(* IEC 61131-3 sources: Yaha/Documentation/Infomaterial/OSCAT/pcworx_basic_333/module_export (part 6) *)

(* ---- SETUP_MONTHS3.ST ---- *)
(*@PROPERTIES_EX@
TYPE: POU
LOCALE: 0
IEC_LANGUAGE: ST
PLC_TYPE: independent
PROC_TYPE: independent
GROUP: SETUP
*)
(*@KEY@:DESCRIPTION*)

(*@KEY@:END_DESCRIPTION*)
FUNCTION_BLOCK SETUP_MONTHS3

(*Group:Default*)

VAR_IN_OUT
	MONTHS3 :	oscat_MONTHS3;
END_VAR

VAR
	init :	BOOL;
END_VAR

(*@KEY@: WORKSHEET
NAME: SETUP_MONTHS3
IEC_LANGUAGE: ST
*)
(* Daten initialisieren *)
IF init THEN RETURN; END_IF;
init := TRUE;

(* ---- english --- *)
MONTHS3[1][01] := 'Jan';
MONTHS3[1][02] := 'Feb';
MONTHS3[1][03] := 'Mar';
MONTHS3[1][04] := 'Apr';
MONTHS3[1][05] := 'May';
MONTHS3[1][06] := 'Jun';
MONTHS3[1][07] := 'Jul';
MONTHS3[1][08] := 'Aug';
MONTHS3[1][09] := 'Sep';
MONTHS3[1][10] := 'Oct';
MONTHS3[1][11] := 'Nov';
MONTHS3[1][12] := 'Dec';

(* ---- german --- *)
MONTHS3[2][01] := 'Jan';
MONTHS3[2][02] := 'Feb';
MONTHS3[2][03] := 'Mrz';
MONTHS3[2][04] := 'Apr';
MONTHs3[2][05] := 'Mai';
MONTHS3[2][06] := 'Jun';
MONTHS3[2][07] := 'Jul';
MONTHS3[2][08] := 'Aug';
MONTHS3[2][09] := 'Sep';
MONTHS3[2][10] := 'Okt';
MONTHS3[2][11] := 'Nov';
MONTHS3[2][12] := 'Dez';

(* ---- french --- *)
MONTHS3[3][01] := 'Jan';
MONTHS3[3][02] := 'Fev';
MONTHS3[3][03] := 'Mar';
MONTHS3[3][04] := 'Avr';
MONTHs3[3][05] := 'Mai';
MONTHS3[3][06] := 'Jun';
MONTHS3[3][07] := 'Jul';
MONTHS3[3][08] := 'Aou';
MONTHS3[3][09] := 'Sep';
MONTHS3[3][10] := 'Oct';
MONTHS3[3][11] := 'Nov';
MONTHS3[3][12] := 'Dec';
(*@KEY@: END_WORKSHEET *)
END_FUNCTION_BLOCK

(* ---- SETUP_WEEKDAYS.ST ---- *)
(*@PROPERTIES_EX@
TYPE: POU
LOCALE: 0
IEC_LANGUAGE: ST
PLC_TYPE: independent
PROC_TYPE: independent
GROUP: SETUP
*)
(*@KEY@:DESCRIPTION*)

(*@KEY@:END_DESCRIPTION*)
FUNCTION_BLOCK SETUP_WEEKDAYS

(*Group:Default*)

VAR_IN_OUT
	WEEKDAYS :	oscat_WEEKDAYS;
END_VAR

VAR
	init :	BOOL;
END_VAR

(*@KEY@: WORKSHEET
NAME: SETUP_WEEKDAYS
IEC_LANGUAGE: ST
*)
(* Daten initialisieren *)
IF init THEN RETURN; END_IF;
init := TRUE;

(* ---- english --- *)
WEEKDAYS[1][01] := 'Monday';
WEEKDAYS[1][02] := 'Tuesday';
WEEKDAYS[1][03] := 'Wednesday';
WEEKDAYS[1][04] := 'Thursday';
WEEKDAYS[1][05] := 'Friday';
WEEKDAYS[1][06] := 'Saturday';
WEEKDAYS[1][07] := 'Sunday';

(* ---- german --- *)
WEEKDAYS[2][01] := 'Montag';
WEEKDAYS[2][02] := 'Dienstag';
WEEKDAYS[2][03] := 'Mittwoch';
WEEKDAYS[2][04] := 'Donnerstag';
WEEKDAYS[2][05] := 'Freitag';
WEEKDAYS[2][06] := 'Samstag';
WEEKDAYS[2][07] := 'Sonntag';

(* ---- french --- *)
WEEKDAYS[3][01] := 'Lundi';
WEEKDAYS[3][02] := 'Mardi';
WEEKDAYS[3][03] := 'Mercredi';
WEEKDAYS[3][04] := 'Jeudi';
WEEKDAYS[3][05] := 'Vendredi';
WEEKDAYS[3][06] := 'Samedi';
WEEKDAYS[3][07] := 'Dimanche';
(*@KEY@: END_WORKSHEET *)
END_FUNCTION_BLOCK

(* ---- SETUP_WEEKDAYS2.ST ---- *)
(*@PROPERTIES_EX@
TYPE: POU
LOCALE: 0
IEC_LANGUAGE: ST
PLC_TYPE: independent
PROC_TYPE: independent
GROUP: SETUP
*)
(*@KEY@:DESCRIPTION*)

(*@KEY@:END_DESCRIPTION*)
FUNCTION_BLOCK SETUP_WEEKDAYS2

(*Group:Default*)

VAR_IN_OUT
	WEEKDAYS2 :	oscat_WEEKDAYS2;
END_VAR

VAR
	init :	BOOL;
END_VAR

(*@KEY@: WORKSHEET
NAME: SETUP_WEEKDAYS2
IEC_LANGUAGE: ST
*)
(* Daten initialisieren *)
IF init THEN RETURN; END_IF;
init := TRUE;

(* ---- english --- *)
WEEKDAYS2[1][01] := 'Mo';
WEEKDAYS2[1][02] := 'Tu';
WEEKDAYS2[1][03] := 'We';
WEEKDAYS2[1][04] := 'Th';
WEEKDAYS2[1][05] := 'Fr';
WEEKDAYS2[1][06] := 'Sa';
WEEKDAYS2[1][07] := 'Su';

(* ---- german --- *)
WEEKDAYS2[2][01] := 'Mo';
WEEKDAYS2[2][02] := 'Di';
WEEKDAYS2[2][03] := 'Mi';
WEEKDAYS2[2][04] := 'Do';
WEEKDAYS2[2][05] := 'Fr';
WEEKDAYS2[2][06] := 'Sa';
WEEKDAYS2[2][07] := 'So';

(* ---- french --- *)
WEEKDAYS2[3][01] := 'Lu';
WEEKDAYS2[3][02] := 'Ma';
WEEKDAYS2[3][03] := 'Me';
WEEKDAYS2[3][04] := 'Je';
WEEKDAYS2[3][05] := 'Ve';
WEEKDAYS2[3][06] := 'Sa';
WEEKDAYS2[3][07] := 'Di';
(*@KEY@: END_WORKSHEET *)
END_FUNCTION_BLOCK

(* ---- SH.ST ---- *)
(*@PROPERTIES_EX@
TYPE: POU
LOCALE: 0
IEC_LANGUAGE: ST
PLC_TYPE: independent
PROC_TYPE: independent
GROUP: ENGINEERING.SIGNAL_PROCESSING
*)
(*@KEY@:DESCRIPTION*)
version 1.1	16 jan 2007
programmer 	hugo
tested by	tobias

this sample and hold module samples an input at the rising edge of clk an stores it in out.
the out stays stable until the next rising clk edge appears.
a trigger output as active for one cycle when the output was updated.
(*@KEY@:END_DESCRIPTION*)
FUNCTION_BLOCK SH

(*Group:Default*)

VAR_INPUT
	IN :	REAL;
	CLK :	BOOL;
END_VAR

VAR_OUTPUT
	OUT :	REAL;
	TRIG :	BOOL;
END_VAR

VAR
	edge :	BOOL;
END_VAR

(*@KEY@: WORKSHEET
NAME: SH
IEC_LANGUAGE: ST
*)
IF clk AND NOT edge THEN
	out := in;
	trig := TRUE;
ELSE;
	trig := FALSE;
END_IF;
edge := clk;

(* revision history

hm 16.1.2007	rev 1.1
	added trig output

*)
(*@KEY@: END_WORKSHEET *)
END_FUNCTION_BLOCK

(* ---- SH_1.ST ---- *)
(*@PROPERTIES_EX@
TYPE: POU
LOCALE: 0
IEC_LANGUAGE: ST
PLC_TYPE: independent
PROC_TYPE: independent
GROUP: ENGINEERING.SIGNAL_PROCESSING
*)
(*@KEY@:DESCRIPTION*)
version 1.2	17 sep 2007
programmer 	hugo
tested by	tobias

this sample and hold module samples an input every PT seconds.
after a ample is taken the output Trig will be active for one cycle.
(*@KEY@:END_DESCRIPTION*)
FUNCTION_BLOCK SH_1

(*Group:Default*)

VAR_INPUT
	IN :	REAL;
	PT :	TIME;
END_VAR

VAR_OUTPUT
	OUT :	REAL;
	TRIG :	BOOL;
END_VAR

VAR
	last :	TIME;
	tx :	TIME;
	T_PLC_MS :	T_PLC_MS;
END_VAR

(*@KEY@: WORKSHEET
NAME: SH_1
IEC_LANGUAGE: ST
*)
(* read system time *)
T_PLC_MS();
tx:= UDINT_TO_TIME(T_PLC_MS.T_PLC_MS);

IF tx - last >= PT THEN
	last := tx;
	out := in;
	trig := TRUE;
ELSE
	trig := FALSE;
END_IF;

(* revision history

HM	6.1.2007	rev 1.1
	added trig output

HM	17.9.2007	rev 1.2
	replaced time() with T_PLC_MS() for compatibility reasons
*)
(*@KEY@: END_WORKSHEET *)
END_FUNCTION_BLOCK

(* ---- SH_2.ST ---- *)
(*@PROPERTIES_EX@
TYPE: POU
LOCALE: 0
IEC_LANGUAGE: ST
PLC_TYPE: independent
PROC_TYPE: independent
GROUP: ENGINEERING.SIGNAL_PROCESSING
*)
(*@KEY@:DESCRIPTION*)
version 1.6	10. mar. 2009
programmer 	hugo
tested by	tobias

this sample and hold module samples an input every PT seconds.
this sample and hold also does avg and other calculations with the input data.
an average is calculated over N samples while for this calculation disc samples are discarded,
disc = 0 all samples are averaged,
if disc = 1 the lowest value is ignored,
if disc = 2 the lowest and highest values are ignored,
and so on.....

(*@KEY@:END_DESCRIPTION*)
FUNCTION_BLOCK SH_2

(*Group:Default*)

VAR_INPUT
	IN :	REAL;
	PT :	TIME;
	N :	INT := INT#16;
	DISC :	INT;
END_VAR

VAR_OUTPUT
	OUT :	REAL;
	TRIG :	BOOL;
	AVG :	REAL;
	HIGH :	REAL;
	LOW :	REAL;
END_VAR

VAR
	M :	INT;
	buf :	oscat_arr_0_15;
	buf2 :	oscat_arr_0_15;
	last :	TIME;
	i :	INT;
	I2 :	INT;
	start :	INT;
	temp :	REAL;
	stop :	INT;
	tx :	TIME;
	d2 :	INT;
	T_PLC_MS :	T_PLC_MS;
END_VAR

(*@KEY@: WORKSHEET
NAME: SH_2
IEC_LANGUAGE: ST
*)
(* read system time *)
T_PLC_MS();
tx:= UDINT_TO_TIME(T_PLC_MS.T_PLC_MS);
d2 := WORD_TO_INT(SHR(INT_TO_WORD(disc),1));

IF tx - last >= PT THEN
	last := tx;
	trig := TRUE;

	(* limit M to 0..16 *)
	M := LIMIT(1,N,16);

	(* edge detected lets take the sample *)
    i := M-1;
    WHILE (i>=1) DO
      i2 := i-1;
      buf2[i] := buf2[i2];
      i:=i-1;
    END_WHILE;

	buf2[0] := in;
	out := in;
	buf := buf2;

	(* sort the ARRAY lowest value AT 0 *)
	FOR start := 0 TO M - 2 DO
		FOR i := start+1 TO M - 1 DO
			IF buf[start] > buf[i] THEN
				temp := buf[start];
				buf[start] := buf[i];
				buf[i] := temp;
			END_IF;
		END_FOR;
	END_FOR;

	(* any calculation with the samples is here *)
	stop := M - 1 - d2;
	start := d2;
	IF NOT even(INT_TO_DINT(disc)) THEN start := start + 1; END_IF;
	avg := 0.0;
	FOR i := start TO stop DO avg := avg + buf[i]; END_FOR;
	avg := avg / INT_TO_REAL(stop - start +1);
	low := buf[start];
	high := buf[stop];
ELSE
	Trig := FALSE;
END_IF;

(* revision history
hm 20. jan. 2007	rev 1.1
	added input N to specify the amout of samples for average and high low calculations
	added trig output

hm 10. sep. 2007 	rev 1.2
	an error would be generated if N was set to 0, now n is forced to1 if set to 0.
	index was out of array.

hm	17. sep. 2007	rev 1.3
	replaced time() with t_plc_ms() for compatibility reasons

hm	6. jan. 2008	rev 1.4
	improved performance

hm	14. jun. 2008	rev 1.5
	set default for input N = 16

hm	10. mar. 2009	rev 1.6
	added type conversion for compatibility reasons

*)
(*@KEY@: END_WORKSHEET *)
END_FUNCTION_BLOCK

(* ---- SH_T.ST ---- *)
(*@PROPERTIES_EX@
TYPE: POU
LOCALE: 0
IEC_LANGUAGE: ST
PLC_TYPE: independent
PROC_TYPE: independent
GROUP: ENGINEERING.SIGNAL_PROCESSING
*)
(*@KEY@:DESCRIPTION*)
version 1.1	18. oct. 2008
programmer 	hugo
tested by	oscat

this sample and hold module samples an input while en is high.
during the high time of en the output follows in.
the out stays stable until the en goes high again.
(*@KEY@:END_DESCRIPTION*)
FUNCTION_BLOCK SH_T

(*Group:Default*)

VAR_INPUT
	IN :	REAL;
	E :	BOOL;
END_VAR

VAR_OUTPUT
	OUT :	REAL;
END_VAR

(*@KEY@: WORKSHEET
NAME: SH_T
IEC_LANGUAGE: ST
*)
IF E THEN out := in; END_IF;

(* revision history
hm	1. sep. 2006	rev 1.0
	original version

hm	18. oct. 2008	rev 1.1
	changed input en to e for compatibility reasons

*)
(*@KEY@: END_WORKSHEET *)
END_FUNCTION_BLOCK

(* ---- SHR_4E.ST ---- *)
(*@PROPERTIES_EX@
TYPE: POU
LOCALE: 0
IEC_LANGUAGE: ST
PLC_TYPE: independent
PROC_TYPE: independent
GROUP: LOGIC.FF_EDGE_TRIGGERED
*)
(*@KEY@:DESCRIPTION*)
version 1.1	25. oct. 2008
programmer 	hugo
tested by	tobias

4 bit shift register with reset
(*@KEY@:END_DESCRIPTION*)
FUNCTION_BLOCK SHR_4E

(*Group:Default*)

VAR_INPUT
	SET :	BOOL;
	D0 :	BOOL;
	CLK :	BOOL;
	RST :	BOOL;
END_VAR

VAR_OUTPUT
	Q0 :	BOOL;
	Q1 :	BOOL;
	Q2 :	BOOL;
	Q3 :	BOOL;
END_VAR

VAR
	trig :	R_TRIG;
END_VAR

(*@KEY@: WORKSHEET
NAME: SHR_4E
IEC_LANGUAGE: ST
*)
(* trig.Q signals a rising edge on clk *)
trig(clk := clk);

IF set OR rst THEN
	Q0 := NOT RST;
	Q1 := Q0;
	Q2 := Q0;
	Q3 := Q0;
ELSIF trig.Q THEN
	Q3 := Q2;
	Q2 := Q1;
	Q1 := Q0;
	Q0 := D0;
END_IF;

(* revision history
hm	4. aug. 2006	rev 1.0
	original version

hm	25. oct. 2008	rev 1.1
	optimized code

*)
(*@KEY@: END_WORKSHEET *)
END_FUNCTION_BLOCK

(* ---- SHR_4UDE.ST ---- *)
(*@PROPERTIES_EX@
TYPE: POU
LOCALE: 0
IEC_LANGUAGE: ST
PLC_TYPE: independent
PROC_TYPE: independent
GROUP: LOGIC.FF_EDGE_TRIGGERED
*)
(*@KEY@:DESCRIPTION*)
version 1.2	14. mar. 2009
programmer 	hugo
tested by	tobias

4 bit shift register with reset up / down direction input
(*@KEY@:END_DESCRIPTION*)
FUNCTION_BLOCK SHR_4UDE

(*Group:Default*)

VAR_INPUT
	SET :	BOOL;
	D0 :	BOOL;
	D3 :	BOOL;
	CLK :	BOOL;
	DN :	BOOL;
	RST :	BOOL;
END_VAR

VAR_OUTPUT
	Q0 :	BOOL;
	Q1 :	BOOL;
	Q2 :	BOOL;
	Q3 :	BOOL;
END_VAR

VAR
	trig :	R_TRIG;
END_VAR

(*@KEY@: WORKSHEET
NAME: SHR_4UDE
IEC_LANGUAGE: ST
*)
(* trig.Q signals a rising edge on clk *)
trig(clk := clk);

IF set OR rst THEN
	Q0 := NOT RST;
	Q1 := Q0;
	Q2 := Q0;
	Q3 := Q0;
ELSIF trig.Q THEN
	IF dn THEN
		Q0 := Q1;
		Q1 := Q2;
		Q2 := Q3;
		Q3 := D3;
	ELSE
		Q3 := Q2;
		Q2 := Q1;
		Q1 := Q0;
		Q0 := D0;
	END_IF;
END_IF;

(* revision history
hm	4. aug. 2006	rev 1.0
	original version

hm	25. oct. 2008	rev 1.1
	optimized code

hm	14. mar. 2009	rev 1.2
	removed double assignments

*)
(*@KEY@: END_WORKSHEET *)
END_FUNCTION_BLOCK

(* ---- SHR_8PLE.ST ---- *)
(*@PROPERTIES_EX@
TYPE: POU
LOCALE: 0
IEC_LANGUAGE: ST
PLC_TYPE: independent
PROC_TYPE: independent
GROUP: LOGIC.FF_EDGE_TRIGGERED
*)
(*@KEY@:DESCRIPTION*)
version 1.0	4 aug 2006
programmer 	hugo
tested by	tobias

8 bit shift register with reset and parallel load
the register can shift up or down
it also has a serial input.
the Din input is on Bit0 for up shift and on bit 7 for down shift
the Dout output is on Bit7 for up shift and on bit 0 for down shift
paralle clock is performed clock synchron while a shift is performed first and then the register is reloaded
(*@KEY@:END_DESCRIPTION*)
FUNCTION_BLOCK SHR_8PLE

(*Group:Default*)

VAR_INPUT
	DIN :	BOOL;
	DLOAD :	BYTE;
	CLK :	BOOL;
	UP :	BOOL := TRUE;
	LOAD :	BOOL;
	RST :	BOOL;
END_VAR

VAR_OUTPUT
	DOUT :	BOOL;
END_VAR

VAR
	edge :	BOOL := TRUE;
	register :	BYTE;
END_VAR

(*@KEY@: WORKSHEET
NAME: SHR_8PLE
IEC_LANGUAGE: ST
*)
(* flankenerkennung clk wird high und edge war high reset ist nicht aktiv und set ist nicht aktiv *)
IF CLK AND edge AND NOT rst THEN
	edge := FALSE;	(* flanke wurde erkannt und weitere flankenerkennung wird verhindert bis edge wieder true ist *)
	(* hier ist der code für das flankenevent *)
	IF UP THEN						(*shift up *)
		register := SHL(register,1);
        register := BIT_LOAD_B(register,Din,0);  (* register.X0 := Din; *)
        Dout     := BIT_OF_DWORD(BYTE_TO_DWORD(register),7);     (* Dout := register.X7; *)
	ELSE						    (* shift down *);
		register := SHR(register,1);
        register := BIT_LOAD_B(register,Din,7);  (* register.X7 := Din; *)
        Dout     := BIT_OF_DWORD(BYTE_TO_DWORD(register),0);     (* Dout := register.X0; *)
	END_IF;
	IF load THEN							(* the byte on Din will be loaded if load = true *)
		register := Dload;
		IF up THEN
            Dout := BIT_OF_DWORD(BYTE_TO_DWORD(register),7); (* register.X7 *)
        ELSE
            Dout := BIT_OF_DWORD(BYTE_TO_DWORD(register),0); (* register.X0 *)
        END_IF;
	END_IF;
END_IF;
IF NOT clk THEN edge := TRUE; END_IF;	(* sobald clk wieder low wird warten auf nächste flanke *)
IF rst THEN									(* wenn reset aktiv dann ausgang rücksetzen *)
	register := BYTE#0;
	Dout := FALSE;
END_IF;
(*@KEY@: END_WORKSHEET *)
END_FUNCTION_BLOCK

(* ---- SHR_8UDE.ST ---- *)
(*@PROPERTIES_EX@
TYPE: POU
LOCALE: 0
IEC_LANGUAGE: ST
PLC_TYPE: independent
PROC_TYPE: independent
GROUP: LOGIC.FF_EDGE_TRIGGERED
*)
(*@KEY@:DESCRIPTION*)
version 1.2	14. mar. 2009
programmer 	hugo
tested by	tobias

8 bit shift register with reset

(*@KEY@:END_DESCRIPTION*)
FUNCTION_BLOCK SHR_8UDE

(*Group:Default*)

VAR_INPUT
	SET :	BOOL;
	D0 :	BOOL;
	D7 :	BOOL;
	CLK :	BOOL;
	DN :	BOOL;
	RST :	BOOL;
END_VAR

VAR_OUTPUT
	Q0 :	BOOL;
	Q1 :	BOOL;
	Q2 :	BOOL;
	Q3 :	BOOL;
	Q4 :	BOOL;
	Q5 :	BOOL;
	Q6 :	BOOL;
	Q7 :	BOOL;
END_VAR

VAR
	trig :	R_TRIG;
END_VAR

(*@KEY@: WORKSHEET
NAME: SHR_8UDE
IEC_LANGUAGE: ST
*)
(* trig.Q signals a rising edge on clk *)
trig(clk := clk);

IF set OR rst THEN
	Q0 := NOT RST;
	Q1 := Q0;
	Q2 := Q0;
	Q3 := Q0;
	Q4 := Q0;
	Q5 := Q0;
	Q6 := Q0;
	Q7 := Q0;
ELSIF trig.Q THEN
	IF dn THEN
		Q0 := Q1;
		Q1 := Q2;
		Q2 := Q3;
		Q3 := Q4;
		Q4 := Q5;
		Q5 := Q6;
		Q6 := Q7;
		Q7 := D7;
	ELSE
		Q7 := Q6;
		Q6 := Q5;
		Q5 := Q4;
		Q4 := Q3;
		Q3 := Q2;
		Q2 := Q1;
		Q1 := Q0;
		Q0 := D0;
	END_IF;
END_IF;

(* revision history
hm	4. aug. 2006	rev 1.0
	original version

hm	25. oct. 2008	rev 1.1
	optimized code

hm	14. mar. 2009	rev 1.2
	removed double assignments

*)
(*@KEY@: END_WORKSHEET *)
END_FUNCTION_BLOCK

(* ---- SIGNAL.ST ---- *)
(*@PROPERTIES_EX@
TYPE: POU
LOCALE: 0
IEC_LANGUAGE: ST
PLC_TYPE: independent
PROC_TYPE: independent
GROUP: ENGINEERING.AUTOMATION
*)
(*@KEY@:DESCRIPTION*)
version 1.0	13 dec 2007
programmer 	hugo
tested by	tobias

this function generates an output signal according to a bit pattern SIG.
the patter is shifted to the output in time steps of TS.
ts defaults to 128 ms if not specified.
(*@KEY@:END_DESCRIPTION*)
FUNCTION_BLOCK SIGNAL

(*Group:Default*)

VAR_INPUT
	IN :	BOOL;
	SIG :	BYTE;
	TS :	TIME;
END_VAR

VAR_OUTPUT
	Q :	BOOL;
END_VAR

VAR
	tx :	DWORD;
	step :	BYTE;
	T_PLC_MS :	T_PLC_MS;
END_VAR

(*@KEY@: WORKSHEET
NAME: SIGNAL
IEC_LANGUAGE: ST
*)
IF in THEN
	(* an alarm is present read system time first *)
    T_PLC_MS();
    tx:= UDINT_TO_DWORD(T_PLC_MS.T_PLC_MS);

	(* calculate the step counter which is the lowest 3 bits of (time / ts) *)
	IF ts > t#0s THEN
		step := DWORD_TO_BYTE(UDINT_TO_DWORD(DWORD_TO_UDINT(tx) / TIME_TO_UDINT(ts)) AND DWORD#16#0000_0007);
	ELSE
		step := DWORD_TO_BYTE(SHR(tx,7) AND DWORD#16#0000_0007);
	END_IF;
	(* convert the value 0-7 in step into one bit only (bit 0-7) *)
	step := SHL(BYTE#1,_BYTE_TO_INT(step));
	(* generate the output signal *)
	Q := (step AND sig) > BYTE#0;
ELSE
	Q := FALSE;
END_IF;

(* revision history
hm	13.12.2007		rev 1.0
	original version

*)
(*@KEY@: END_WORKSHEET *)
END_FUNCTION_BLOCK

(* ---- SIGNAL_4.ST ---- *)
(*@PROPERTIES_EX@
TYPE: POU
LOCALE: 0
IEC_LANGUAGE: ST
PLC_TYPE: independent
PROC_TYPE: independent
GROUP: ENGINEERING.AUTOMATION
*)
(*@KEY@:DESCRIPTION*)
version 1.0	13 dec 2007
programmer 	hugo
tested by	tobias

this function generates one out of 4 signals specified by bit patterns S1 .. S4.
the selected pattern will be shifted with the step time TS.
In1 has higher priority then In2 which has higher priority then IN3 and in4 has the lowest priority.
ts defaults to 128 ms if not specified.
(*@KEY@:END_DESCRIPTION*)
FUNCTION_BLOCK SIGNAL_4

(*Group:Default*)

VAR_INPUT
	IN1 :	BOOL;
	IN2 :	BOOL;
	IN3 :	BOOL;
	IN4 :	BOOL;
	TS :	TIME;
	S1 :	BYTE := 2#1111_1111;
	S2 :	BYTE := 2#1111_0000;
	S3 :	BYTE := 2#1010_1010;
	S4 :	BYTE := 2#1010_0000;
END_VAR

VAR_OUTPUT
	Q :	BOOL;
END_VAR

VAR
	sig :	signal;
END_VAR

(*@KEY@: WORKSHEET
NAME: SIGNAL_4
IEC_LANGUAGE: ST
*)
(* an alarm is present read system time first *)
(* check if an alarm is present if yes set sig to the alarm pattern otherwise exit the routine *)
IF in1 THEN
	sig(in := TRUE, sig := s1, TS := TS);
ELSIF in2 THEN
	sig(in := TRUE, sig := s2, TS := TS);
ELSIF in3 THEN
	sig(in := TRUE, sig := s3, TS := TS);
ELSIF in4 THEN
	sig(in := TRUE, sig := s4, TS := TS);
ELSE
	sig(in := FALSE);
END_IF;

(* set the output *)
Q := sig.Q;

(* revision history
hm	13.12.2007		rev 1.0
	original version

*)
(*@KEY@: END_WORKSHEET *)
END_FUNCTION_BLOCK

(* ---- SPEED.ST ---- *)
(*@PROPERTIES_EX@
TYPE: POU
LOCALE: 0
IEC_LANGUAGE: ST
PLC_TYPE: independent
PROC_TYPE: independent
GROUP: ENGINEERING.CONVERSION
*)
(*@KEY@:DESCRIPTION*)
version 1.1	11. mar. 2009
programmer 	hugo
tested by	oscat

this function converts different speed units
any unused input can simply be left open.
different inputs connected at the same time will be added up.
(*@KEY@:END_DESCRIPTION*)
FUNCTION_BLOCK SPEED

(*Group:Default*)

VAR_INPUT
	MS :	REAL;
	KMH :	REAL;
	KN :	REAL;
	MH :	REAL;
END_VAR

VAR_OUTPUT
	YMS :	REAL;
	YKMH :	REAL;
	YKN :	REAL;
	YMH :	REAL;
END_VAR

(*@KEY@: WORKSHEET
NAME: SPEED
IEC_LANGUAGE: ST
*)
Yms := ms +
		kmh * 0.27777777777778 +
		kn * 0.5144444 +
		mh * 0.44704;
Ykmh := Yms * 3.6;
Ykn := Yms * 1.94384466037535;
Ymh := Yms * 2.23693629205440;

(*
Geschwindigkeit Meter durch Sekunde m/s 1 m/s = 3,6 km/h
km durch (pro) Stunde, nicht „Stundenkilometer“ verwenden
Knoten kn 1 kn = 1 sm/h = 0,5144 m/s

*)
(*@KEY@: END_WORKSHEET *)
END_FUNCTION_BLOCK

(* ---- SRAMP.ST ---- *)
(*@PROPERTIES_EX@
TYPE: POU
LOCALE: 0
IEC_LANGUAGE: ST
PLC_TYPE: independent
PROC_TYPE: independent
GROUP: ENGINEERING.AUTOMATION
*)
(*@KEY@:DESCRIPTION*)
version 1.1	11. mar. 2009
programmer 	hugo
tested by	tobias

RAMPS generates output signal which are slew rate and acceleration controlled.

(*@KEY@:END_DESCRIPTION*)
FUNCTION_BLOCK SRAMP

(*Group:Default*)

VAR_INPUT
	X :	REAL;
	A_UP :	REAL;
	A_DN :	REAL;
	VU_MAX :	REAL;
	VD_MAX :	REAL;
	LIMIT_HIGH :	REAL;
	LIMIT_LOW :	REAL;
	RST :	BOOL;
END_VAR

VAR_OUTPUT
	Y :	REAL;
	V :	REAL;
END_VAR

VAR
	cycle_time :	TC_S;
	init :	BOOL;
END_VAR

(*@KEY@: WORKSHEET
NAME: SRAMP
IEC_LANGUAGE: ST
*)
(* read the system_time in microseconds *)
cycle_time();

(* assure range of inputs *)
A_up := MAX(0.0,A_UP);
A_dn := MIN(0.0,A_dn);
VU_max := MAX(0.0,VU_max);
VD_max := MIN(0.0,VD_MAX);

(* calculate the output offset *)
IF rst OR NOT init THEN
	init := TRUE;
	Y := 0.0;
	V := 0.0;
ELSIF X = Y THEN
	v := 0.0;
ELSIF X > Y THEN
	(* output is too low >> ramp up and brake at the end *)
	(* accelerate the speed and limit to vu_max *)
	v := MIN(v + A_UP * cycle_time.TC, vu_max);
	(* calculate the max speed to be able to brake and select the lowest *)
	v := MIN(SQRT((Y-X) * 2.0 * A_DN), v);
	(* calculate the output and obey limits *)
	y := LIMIT(limit_low, y + MIN(v * cycle_time.TC, X-Y), limit_high);
ELSIF X < Y THEN
	(* output is too high >> ramp dn and brake at the end *)
	(* accelerate the speed and limit to vd_max *)
	v := MAX(v + A_DN * cycle_time.TC, vd_max);
	(* calculate the max speed to be able to brake and select the lowest *)
	v := MAX(-SQRT((Y-X) * 2.0 * A_UP), v);
	(* calculate the output and obey limits *)
	y := LIMIT(limit_low, y + MAX(v * cycle_time.TC, X-Y), limit_high);
END_IF;

(* revision history
hm	13. mar. 2008	rev 1.0
	original version

hm	11. mar. 2009	rev 1.1
	real constants updated to new systax using dot

*)

(*@KEY@: END_WORKSHEET *)
END_FUNCTION_BLOCK

(* ---- STACK_16.ST ---- *)
(*@PROPERTIES_EX@
TYPE: POU
LOCALE: 0
IEC_LANGUAGE: ST
PLC_TYPE: independent
PROC_TYPE: independent
GROUP: LOGIC.MEMORY
*)
(*@KEY@:DESCRIPTION*)
version 2.0	25. jul 2009
programmer 	hugo
tested by	oscat

16 Dword STACK memory

(*@KEY@:END_DESCRIPTION*)
FUNCTION_BLOCK STACK_16

(*Group:Default*)

VAR_INPUT
	DIN :	DWORD;
	E :	BOOL := TRUE;
	RD :	BOOL;
	WD :	BOOL;
	RST :	BOOL;
END_VAR

VAR_OUTPUT
	DOUT :	DWORD;
	EMPTY :	BOOL := TRUE;
	FULL :	BOOL;
END_VAR

VAR
	pt :	INT;
	stack :	oscat_ardw_0_15;
END_VAR

(*@KEY@: WORKSHEET
NAME: STACK_16
IEC_LANGUAGE: ST
*)
IF RST THEN
	(* asynchronous reset for the fifo *)
	pt := 0;
	EMPTY := TRUE;
	FULL := FALSE;
	Dout := DWORD#0;
ELSIF E THEN
	IF NOT EMPTY AND RD THEN
		(* read one element *)
		pt := pt - 1;
		Dout := stack[pt];
		EMPTY := pt = 0;
		FULL := FALSE;
	END_IF;
	IF NOT FULL AND WD THEN
		(* write one element *)
		stack[pt] := Din;
		pt := pt + 1;
		FULL := pt > 15;
		EMPTY := FALSE;
	END_IF;
END_IF;

(* revision history
hm	4. aug. 2006	rev 1.0
	original version

hm	19. feb 2008	rev 1.1
	performance improvements

hm	17. oct. 2008	rev 1.2
	deleted unnecessary init with 0

hm	27. oct. 2008	rev 1.3
	optimized performance

hm	25. jul 2009	rev 2.0
	changed inputs to allow simultsaneous read and write
*)

(*@KEY@: END_WORKSHEET *)
END_FUNCTION_BLOCK

(* ---- STACK_32.ST ---- *)
(*@PROPERTIES_EX@
TYPE: POU
LOCALE: 0
IEC_LANGUAGE: ST
PLC_TYPE: independent
PROC_TYPE: independent
GROUP: LOGIC.MEMORY
*)
(*@KEY@:DESCRIPTION*)
version 2.0	25. jul 2009
programmer 	hugo
tested by	oscat

32 Dword STACK memory
(*@KEY@:END_DESCRIPTION*)
FUNCTION_BLOCK STACK_32

(*Group:Default*)

VAR_INPUT
	DIN :	DWORD;
	E :	BOOL := TRUE;
	RD :	BOOL;
	WD :	BOOL;
	RST :	BOOL;
END_VAR

VAR_OUTPUT
	DOUT :	DWORD;
	EMPTY :	BOOL := TRUE;
	FULL :	BOOL;
END_VAR

VAR
	pt :	INT;
	stack :	oscat_ardw_0_31;
END_VAR

(*@KEY@: WORKSHEET
NAME: STACK_32
IEC_LANGUAGE: ST
*)
IF RST THEN
	(* asynchronous reset for the fifo *)
	pt := 0;
	EMPTY := TRUE;
	FULL := FALSE;
	Dout := DWORD#0;
ELSIF E THEN
	IF NOT EMPTY AND RD THEN
		(* read one element *)
		pt := pt - 1;
		Dout := stack[pt];
		EMPTY := pt = 0;
		FULL := FALSE;
	END_IF;
	IF NOT FULL AND WD THEN
		(* write one element *)
		stack[pt] := Din;
		pt := pt + 1;
		FULL := pt > 31;
		EMPTY := FALSE;
	END_IF;
END_IF;

(* revision history
hm	4. aug. 2006	rev 1.0
	original version

hm	19. feb 2008	rev 1.1
	performance improvements

hm	17. oct. 2008	rev 1.2
	deleted unnecessary init with 0

ks	27. oct. 2008	rev 1.3
	optimized performance

hm	25. jul 2009	rev 2.0
	changed inputs to allow simultsaneous read and write

*)

(*@KEY@: END_WORKSHEET *)
END_FUNCTION_BLOCK

(* ---- STAIR2.ST ---- *)
(*@PROPERTIES_EX@
TYPE: POU
LOCALE: 0
IEC_LANGUAGE: ST
PLC_TYPE: independent
PROC_TYPE: independent
GROUP: ENGINEERING.SIGNAL_PROCESSING
*)
(*@KEY@:DESCRIPTION*)
version 1.4	10. mar. 2009
programmer 	hugo
tested by	oscat

the function stair2 converts an anlog input signal to a staircase like output.
D is the step width for the output signal. the output will use D as a hysteresis for a stairchange.
if D = 0 then the output follows the input without a chage.
(*@KEY@:END_DESCRIPTION*)
FUNCTION_BLOCK STAIR2

(*Group:Default*)

VAR_INPUT
	X :	REAL;
	D :	REAL;
END_VAR

VAR_OUTPUT
	Y :	REAL;
END_VAR

(*@KEY@: WORKSHEET
NAME: STAIR2
IEC_LANGUAGE: ST
*)
IF D > 0.0 THEN
	IF X >= Y + D OR X <= Y - D THEN Y := INT_TO_REAL(FLOOR(X/D)) * D; END_IF;
ELSE
	Y := X;
END_IF;

(* revision history
hm	28 jan 2007		rev 1.0
	original version

hm	27. dec 2007	rev 1.1
	changed code for better performance

hm	30. jun. 2008	rev 1.2
	added type conversions to avoid warnings under codesys 3.0

ks	26. oct. 2008	rev 1.3
	improved code

hm	10. mar. 2009	rev 1.4
	real constants updated to new systax using dot

*)
(*@KEY@: END_WORKSHEET *)
END_FUNCTION_BLOCK

(* ---- STATUS_TO_ESR.ST ---- *)
(*@PROPERTIES_EX@
TYPE: POU
LOCALE: 0
IEC_LANGUAGE: ST
PLC_TYPE: independent
PROC_TYPE: independent
GROUP: OTHER
*)
(*@KEY@:DESCRIPTION*)
version 1.0	6 oct 2006
programmer 	hugo
tested by	tobias

status_to_esr creates esr data from a status byte.
(*@KEY@:END_DESCRIPTION*)
FUNCTION_BLOCK STATUS_TO_ESR

(*Group:Default*)

VAR_INPUT
	STATUS :	BYTE;
	ADRESS :	oscat_STRING10;
	DT_IN :	UDINT;
	TS :	TIME;
END_VAR

VAR_OUTPUT
	STATUS_TO_ESR :	oscat_esr_data;
END_VAR

(*@KEY@: WORKSHEET
NAME: STATUS_TO_ESR
IEC_LANGUAGE: ST
*)
IF status < BYTE#100 THEN
	status_to_ESR.typ := BYTE#1;
ELSIF status < BYTE#200 THEN
	status_to_ESR.typ := BYTE#2;
ELSE
	status_to_ESR.typ := BYTE#3;
END_IF;
status_to_ESR.adress:= adress;
status_to_ESR.DS := DT_in;
status_to_ESR.TS := TS;
status_to_ESR.data[0] := status;
(*@KEY@: END_WORKSHEET *)
END_FUNCTION_BLOCK

(* ---- STORE_8.ST ---- *)
(*@PROPERTIES_EX@
TYPE: POU
LOCALE: 0
IEC_LANGUAGE: ST
PLC_TYPE: independent
PROC_TYPE: independent
GROUP: LOGIC.FF_PULSE_TRIGGERED
*)
(*@KEY@:DESCRIPTION*)
version 1.2	14. mar. 2009
programmer 	hugo
tested by	oscat

Store_4 stores up to 4 boolean inputs until a reset is clearing the outputs.
the respective output is set with a true at the respective input and stays true until a reset is generated.
a set input is used to set all outputs true at the same time, independent of their inputs.
a clear input is used to reset only the lowest priority of the outputs one at a time.
the lowest priority is q3.
(*@KEY@:END_DESCRIPTION*)
FUNCTION_BLOCK STORE_8

(*Group:Default*)

VAR_INPUT
	SET :	BOOL;
	D0 :	BOOL;
	D1 :	BOOL;
	D2 :	BOOL;
	D3 :	BOOL;
	D4 :	BOOL;
	D5 :	BOOL;
	D6 :	BOOL;
	D7 :	BOOL;
	CLR :	BOOL;
	RST :	BOOL;
END_VAR

VAR_OUTPUT
	Q0 :	BOOL;
	Q1 :	BOOL;
	Q2 :	BOOL;
	Q3 :	BOOL;
	Q4 :	BOOL;
	Q5 :	BOOL;
	Q6 :	BOOL;
	Q7 :	BOOL;
END_VAR

VAR
	edge :	BOOL;
END_VAR

(*@KEY@: WORKSHEET
NAME: STORE_8
IEC_LANGUAGE: ST
*)
IF rst OR set THEN
	q0 := NOT rst;
	q1 := q0;
	q2 := q0;
	q3 := q0;
	q4 := q0;
	q5 := q0;
	q6 := q0;
	q7 := q0;
ELSE
	IF D0 THEN Q0 := TRUE; END_IF;
	IF D1 THEN Q1 := TRUE; END_IF;
	IF D2 THEN Q2 := TRUE; END_IF;
	IF D3 THEN Q3 := TRUE; END_IF;
	IF D4 THEN Q4 := TRUE; END_IF;
	IF D5 THEN Q5 := TRUE; END_IF;
	IF D6 THEN Q6 := TRUE; END_IF;
	IF D7 THEN Q7 := TRUE; END_IF;

	IF clr AND NOT edge THEN
		IF q0 THEN q0 := FALSE;
		ELSIF q1 THEN q1 := FALSE;
		ELSIF q2 THEN q2 := FALSE;
		ELSIF q3 THEN q3 := FALSE;
		ELSIF q4 THEN q4 := FALSE;
		ELSIF q5 THEN q5 := FALSE;
		ELSIF q6 THEN q6 := FALSE;
		ELSE q7 := FALSE;
		END_IF;
	END_IF;
	edge := clr;
END_IF;

(* revision history
hm	25.12.2007	rev 1.0
	original version

hm	30. oct. 2008	rev 1.1
	optimized performance

hm	14. mar. 2009	rev 1.2
	removed double assignments

*)

(*@KEY@: END_WORKSHEET *)
END_FUNCTION_BLOCK

(* ---- STRING_TO_TOD.ST ---- *)
(*@PROPERTIES_EX@
TYPE: POU
LOCALE: 0
IEC_LANGUAGE: ST
PLC_TYPE: independent
PROC_TYPE: independent
GROUP: EMULATION
*)
(*@KEY@:DESCRIPTION*)

(*@KEY@:END_DESCRIPTION*)
FUNCTION_BLOCK STRING_TO_TOD

(*Group:Default*)

VAR_INPUT
	_TOD :	STRING;
END_VAR

VAR_OUTPUT
	STRING_TO_TOD :	UDINT;
END_VAR

VAR
	pos :	INT;
	i :	INT;
	tmp :	STRING;
	tmp2 :	STRING;
END_VAR

(*@KEY@: WORKSHEET
NAME: STRING_TO_TOD
IEC_LANGUAGE: ST
*)
(*
TIME_OF_DAY-Konstanten, zum Speichern von Uhrzeiten:

Eine TIME_OF_DAY-Deklaration beginnt mit "tod#", "TOD#", "TIME_OF_DAY#"
oder "time_of_day#", anschließend können Sie eine Uhrzeit angeben in der Schreibweise:
Stunde:Minute:Sekunde. Sekunden können dabei als reelle Zahlen angegeben werden,
es können also auch Sekundenbruchteile angegeben werden.
Mögliche Werte: 00:00:00 bis 23:59:59.999.

Beispiele:

TIME_OF_DAY#15:36:30.123

tod#00:00:00
*)

STRING_TO_TOD := UDINT#0;
i := LEN(_TOD);
pos :=FIND(_TOD,'#');

IF pos>0 AND i>pos THEN
  tmp := RIGHT(_TOD,LEN(_TOD)-pos);
  pos := FIND(tmp,':');
  IF pos>1 THEN
    tmp2 := LEFT(tmp,pos-1);
    tmp := RIGHT(tmp,LEN(tmp)-pos);
    STRING_TO_TOD := STRING_TO_UDINT(tmp2) * UDINT#3600000;

    pos :=FIND(tmp,':');
    IF pos>1 THEN
      tmp2 := LEFT(tmp,pos-1);
      tmp := RIGHT(tmp,LEN(tmp)-pos);
      STRING_TO_TOD := STRING_TO_TOD + STRING_TO_UDINT(tmp2) * UDINT#60000;

      STRING_TO_TOD := STRING_TO_TOD + STRING_TO_UDINT(tmp) * UDINT#1000;
    END_IF;
  END_IF;
END_IF;
(*@KEY@: END_WORKSHEET *)
END_FUNCTION_BLOCK

(* ---- SUN_POS.ST ---- *)
(*@PROPERTIES_EX@
TYPE: POU
LOCALE: 0
IEC_LANGUAGE: ST
PLC_TYPE: independent
PROC_TYPE: independent
GROUP: TIME_DATE
*)
(*@KEY@:DESCRIPTION*)
version 2.1	7. mar. 2009
programmer 	hugo
tested by		oscat

this FUNCTION block calculates the sun position for a given date and time.
the times are calculated in utc and have to be corrected for the given time zone.
B is the angle from north and HR is the highth in degrees.

(*@KEY@:END_DESCRIPTION*)
FUNCTION_BLOCK SUN_POS

(*Group:Default*)

VAR_INPUT
	LATITUDE :	REAL;(*latitude of geographical position*)
	LONGITUDE :	REAL;(*longitude of geographical position*)
	UTC :	UDINT;(*world time*)
END_VAR

VAR_OUTPUT
	B :	REAL;
	HR :	REAL;
END_VAR

VAR
	g :	REAL;
	a :	REAL;
	d :	REAL;
	h :	REAL;
	t1 :	REAL;
	n :	REAL;
	e :	REAL;
	c :	REAL;
	tau :	REAL;
	sin_d :	REAL;
	rlat :	REAL;
	sin_lat :	REAL;
	cos_lat :	REAL;
	cos_tau :	REAL;
	cos_d :	REAL;
	MATH_PI :	REAL := 3.14159265358979323846264338327950288;
	MATH_PI2 :	REAL := 6.28318530717958647692528676655900576;
END_VAR

(*@KEY@: WORKSHEET
NAME: SUN_POS
IEC_LANGUAGE: ST
*)
(* EXIT the routine IF it was executed within 10 seconds which is equal to 0.04 degrees accuracy
depending on startup conditions this could lead to a lockup for 10 seconds and not delivering a usable position
tx := T_PLC_MS();
IF tx - last < 10000 THEN RETURN; END_IF;
last := tx;
*)

(* n is the julian date and the number of days since 1.1.2000-12:00 midday *)
(* be careful for step7 date startes 1.1.1990 instead of 1.1.1970 *)
(* for step7 this line must change *)
n := UDINT_TO_REAL(UTC - UDINT#946728000) * 0.000011574074074074;
g :=MODR(6.240040768 + 0.01720197 * n, MATH_PI2);
d := MODR(4.89495042 + 0.017202792 * n, MATH_PI2) + 0.033423055 * SIN(g) + 0.000349066 * SIN(2.0*g);
e := 0.409087723 - 0.000000006981317008 * n;
cos_d := COS(d);
sin_d := SIN(d);
a := ATAN(COS(e) * sin_d / cos_d);
IF cos_d < 0.0 THEN a := a + MATH_PI; END_IF;
c := ASIN(SIN(e) * sin_d);

(* also here we must be very careful utc is from 1.1.1970 for step7 the formula must change *)
tau := RAD(MODR(6.697376 + (n - 0.25) * 0.0657098245037645 + TOD_TO_REAL(DT_TO_TOD(utc)) * 0.0000002785383333, 24.0) * 15.0 + longitude) - a;
rlat := RAD(latitude);
sin_lat := SIN(rlat);
cos_lat := COS(rlat);
cos_tau := COS(tau);
t1 := cos_tau * sin_lat - TAN(c) * cos_lat;
B := ATAN(SIN(tau) / t1);
IF t1 < 0.0 THEN B := B + MATH_PI2; ELSE B := B + MATH_PI; END_IF;
B := DEG(MODR(B, MATH_PI2));
h := DEG(ASIN(COS(C) * cos_tau * cos_lat +SIN(c) * sin_lat));
IF h > 180.0 THEN h := h - 360.0; END_IF;
(* consider refraction *)
HR := h + REFRACTION(h);

(* revision history
hm	1. feb 2007	rev 1.0
	original version

hm	6. jan 2008	rev 1.1
	performance improvements

hm	18. jan 2008	rev 1.2
	further performance improvements
	only calculate once every 10 seconds

hm	16. mar. 2008	rev 1.3
	added type conversion to avoid warnings under codesys 3.0

hm	30. jun. 2008	rev 1.4
	added type conversions to avoid warnings under codesys 3.0

hm	18. oct. 2008	rev 1.5
	using math constants

hm	17. dec. 2008	rev 1.6
	angles below horizon are displayed in negative degrees

hm	27. feb. 2009	rev 2.0
	new code with better accuracy

hm	7. mar. 2009	rev 2.1
	refraction is added after angle normalization
	deleted 10 second lockout
	added output for astronomical heigth h
*)
(*@KEY@: END_WORKSHEET *)
END_FUNCTION_BLOCK

(* ---- SUN_TIME.ST ---- *)
(*@PROPERTIES_EX@
TYPE: POU
LOCALE: 0
IEC_LANGUAGE: ST
PLC_TYPE: independent
PROC_TYPE: independent
GROUP: TIME_DATE
*)
(*@KEY@:DESCRIPTION*)
version 1.7	25. jan. 2011
programmer 	hugo
tested by	tobias

this FUNCTION block calculates the sun rise, sun set, sun offset at midday sun declination for a given date
for performance reasons the algorithm has been simplified and is accurate within a few minutes only
the times are calculated in utc and have to be corrected for the given time zone
this correction is not done within sun_time because it would be a problem on days where dst is enabled or disabled

(*@KEY@:END_DESCRIPTION*)
FUNCTION_BLOCK SUN_TIME

(*Group:Default*)

VAR_INPUT
	LATITUDE :	REAL;(*latitude of geographical position*)
	LONGITUDE :	REAL;(*longitude of geographical position*)
	UTC :	UDINT;(*world time*)
	H :	REAL := -0.83333333333;(*heighth above horizon for sunrise*)
END_VAR

VAR_OUTPUT
	MIDDAY :	UDINT;(*astrological midday in hours when sun stand at south direction*)
	SUN_RISE :	UDINT;(*sun rise for current day in local time*)
	SUN_SET :	UDINT;(*sun set for current day in local time*)
	SUN_DECLINATION :	REAL;(*sun declination at midday in degrees*)
END_VAR

VAR
	DK :	REAL;(*sun declination at midday*)
	delta :	UDINT;(*delta from midday for sunrise and sunset*)
	B :	REAL;
END_VAR

(*@KEY@: WORKSHEET
NAME: SUN_TIME
IEC_LANGUAGE: ST
*)
B := latitude * 0.0174532925199433;
MIDDAY := SUN_MIDDAY(longitude, utc);
DK := 0.40954 * SIN(0.0172 * (INT_TO_REAL(DAY_OF_YEAR(utc)) - 79.35));
sun_declination := DEG(DK);
IF sun_declination > 180.0 THEN sun_declination := sun_declination - 360.0; END_IF;
sun_declination := 90.0 - LATITUDE + sun_declination;
delta := TIME_TO_UDINT(HOUR_TO_TIME(ACOS((SIN(RAD(H)) - SIN(B) * SIN(DK)) / (COS(B) * COS(DK))) * 3.819718632));
sun_rise := MIDDAY - delta;
sun_set := MIDDAY + delta;

(* revision history

rev 1.1	hm	20.1.2007
	deleted unused variables sun_riseR and sun_setR

rev 1.2 hm 17.4.2007
	corrected error while sun:midday would not be corrected for longitude.

rev 1.3	hm	6. jan 2008
	performance improvements

rev	1.4 hm	17. jan 2008
	calculation is now only performed once a day

hm	10. mar. 2009	rev 1.5
	improved performance
	calculation will be performed on every call to allow movong installations

hm	26. jul 2009	rev 1.6
	fixed a problem with wrong midday calculation

hm	25. jan. 2011	rev 1.7
	using function sun_midday
	corrected angle of sun_declination
	added input H
*)
(*@KEY@: END_WORKSHEET *)
END_FUNCTION_BLOCK

(* ---- T_PLC_MS.ST ---- *)
(*@PROPERTIES_EX@
TYPE: POU
LOCALE: 0
IEC_LANGUAGE: ST
PLC_TYPE: independent
PROC_TYPE: independent
GROUP: ENGINEERING.MEASUREMENTS
*)
(*@KEY@:DESCRIPTION*)
version 1.1	12 nov 2007
programmer 	hugo
tested by	tobias

T_PLC_MS reads the internal PLC timer and return the time, it has the advantage to be able to set a debug mode
and speed up the counter to test the plc timer overrun which occurs every 50 days respectively 25 days at siemens S7
this routine also allows to correct the behavior of s7 where the internal plc counter will not count all 32 bits.
(*@KEY@:END_DESCRIPTION*)
FUNCTION_BLOCK T_PLC_MS

(*Group:Default*)

VAR_OUTPUT
	T_PLC_MS :	UDINT;
END_VAR

VAR_EXTERNAL
	PLC_TICKS_PER_SEC :	INT;(*Systemticks pro Sekunde*)
	PLC_SYS_TICK_CNT :	DINT;(*Anzahl der Systemticks*)
END_VAR

(*Group:Debug-Parameter*)

VAR
	debug :	BOOL;(*Debug-Mode ON / OFF*)
	N :	INT;(*Debug-Faktor*)
	Offset :	UDINT;(*Debug-Offset*)
	temp :	DWORD := DWORD#1;(*Debug-Offset*)
	mode :	BOOL;(*modus*)
	faktor :	UDINT;(*Systemtakt-Faktor*)
	init :	BOOL;
	v_plc_ticks_per_sec :	UDINT;
	base :	UDINT := UDINT#1000;
END_VAR

(*@KEY@: WORKSHEET
NAME: T_PLC_MS
IEC_LANGUAGE: ST
*)
IF init = FALSE THEN
	v_plc_ticks_per_sec := INT_TO_UDINT(PLC_TICKS_PER_SEC);
	IF v_plc_ticks_per_sec = UDINT#1024 THEN
		faktor := UDINT#1;
		mode := FALSE;
	ELSIF v_plc_ticks_per_sec > UDINT#0 THEN
		IF v_plc_ticks_per_sec <= base THEN
			faktor := base / v_plc_ticks_per_sec;
			mode := FALSE;
		ELSE
			faktor := v_plc_ticks_per_sec / base;
			mode := TRUE;
		END_IF;
	ELSE
		faktor := UDINT#1;
	END_IF;
	init := TRUE;
END_IF;

IF mode THEN
	T_PLC_MS := DINT_TO_UDINT(PLC_SYS_TICK_CNT) / faktor;
ELSE
	T_PLC_MS := DINT_TO_UDINT(PLC_SYS_TICK_CNT) * faktor;
END_IF;

IF debug THEN
	T_PLC_MS := (DWORD_TO_UDINT(SHL(UDINT_TO_DWORD(T_PLC_MS),N) OR SHL(temp,N)) - UDINT#1) + Offset;
END_IF;

(* revision history
hm	14.9.2007	rev 1.0
	original version

hm	12. nov 2007	rev 1.1
	added temporaray variable tx because some compilers could not handle time() as an argument

*)
(*@KEY@: END_WORKSHEET *)
END_FUNCTION_BLOCK

(* ---- T_PLC_US.ST ---- *)
(*@PROPERTIES_EX@
TYPE: POU
LOCALE: 0
IEC_LANGUAGE: ST
PLC_TYPE: independent
PROC_TYPE: independent
GROUP: ENGINEERING.MEASUREMENTS
*)
(*@KEY@:DESCRIPTION*)
version 1.1	12 nov 2007
programmer 	hugo
tested by	tobias

T_PLC_US reads the internal PLC timer and return the time, it has the advantage to be able to set a debug mode
and speed up the counter to test the plc timer overrun which occurs every 50 days respectively 25 days at siemens S7
this routine also allows to correct the behavior of s7 where the internal plc counter will not count all 32 bits.
(*@KEY@:END_DESCRIPTION*)
FUNCTION_BLOCK T_PLC_US

(*Group:Default*)

VAR_OUTPUT
	T_PLC_US :	UDINT;
END_VAR

VAR_EXTERNAL
	PLC_TICKS_PER_SEC :	INT;(*Systemticks pro Sekunde*)
	PLC_SYS_TICK_CNT :	DINT;(*Anzahl der Systemticks*)
END_VAR

(*Group:Debug-Parameter*)

VAR
	debug :	BOOL;(*Debug-Mode ON / OFF*)
	N :	INT;(*Debug-Faktor*)
	Offset :	UDINT;(*Debug-Offset*)
	temp :	DWORD := DWORD#1;(*Debug-Offset*)
	mode :	BOOL;(*modus*)
	faktor :	UDINT;(*Systemtakt-Faktor*)
	init :	BOOL;
	v_plc_ticks_per_sec :	UDINT;
	base :	UDINT := UDINT#1000000;
END_VAR

(*@KEY@: WORKSHEET
NAME: T_PLC_US
IEC_LANGUAGE: ST
*)
IF init = FALSE THEN
	v_plc_ticks_per_sec := INT_TO_UDINT(PLC_TICKS_PER_SEC);
	IF v_plc_ticks_per_sec = UDINT#1024 THEN
		faktor := UDINT#1000;
		mode := FALSE;
	ELSIF v_plc_ticks_per_sec > UDINT#0 THEN
		IF v_plc_ticks_per_sec <= base THEN
			faktor := base / v_plc_ticks_per_sec;
			mode := FALSE;
		ELSE
			faktor := v_plc_ticks_per_sec / base;
			mode := TRUE;
		END_IF;
	ELSE
		faktor := UDINT#1;
	END_IF;
	init := TRUE;
END_IF;

IF mode THEN
	T_PLC_US := DINT_TO_UDINT(PLC_SYS_TICK_CNT) / faktor;
ELSE
	T_PLC_US := DINT_TO_UDINT(PLC_SYS_TICK_CNT) * faktor;
END_IF;

IF debug THEN
	T_PLC_US := (DWORD_TO_UDINT(SHL(UDINT_TO_DWORD(T_PLC_US),N) OR SHL(temp,N)) - UDINT#1) + Offset;
END_IF;

(* revision history
hm	14.9.2007	rev 1.0
	original version

hm	12. nov 2007	rev 1.1
	added temporaray variable tx because some compilers could not handle time() as an argument

*)
(*@KEY@: END_WORKSHEET *)
END_FUNCTION_BLOCK

(* ---- TC_MS.ST ---- *)
(*@PROPERTIES_EX@
TYPE: POU
LOCALE: 0
IEC_LANGUAGE: ST
PLC_TYPE: independent
PROC_TYPE: independent
GROUP: ENGINEERING.MEASUREMENTS
*)
(*@KEY@:DESCRIPTION*)
version 1.0	13 mar 2008
programmer 	hugo
tested by	tobias

TC_MS delivers the time it was last called on the output TC in Milliseconds.
(*@KEY@:END_DESCRIPTION*)
FUNCTION_BLOCK TC_MS

(*Group:Default*)

VAR_OUTPUT
	TC :	DWORD;
END_VAR

VAR
	init :	BOOL;
	tx :	UDINT;
	last :	UDINT;
	T_PLC_MS :	T_PLC_MS;
END_VAR

(*@KEY@: WORKSHEET
NAME: TC_MS
IEC_LANGUAGE: ST
*)
(* read system time and prepare input data *)
T_PLC_MS();
tx:= T_PLC_MS.T_PLC_MS;

IF NOT init THEN
	init := TRUE;
	TC := DWORD#0;
ELSE
	tc := UDINT_TO_DWORD(tx - last);
END_IF;
last := tx;

(* revision history
hm		13. mar. 2008	rev 1.0
	original version

*)
(*@KEY@: END_WORKSHEET *)
END_FUNCTION_BLOCK

(* ---- TC_S.ST ---- *)
(*@PROPERTIES_EX@
TYPE: POU
LOCALE: 0
IEC_LANGUAGE: ST
PLC_TYPE: independent
PROC_TYPE: independent
GROUP: ENGINEERING.MEASUREMENTS
*)
(*@KEY@:DESCRIPTION*)
version 1.2	11. mar. 2009
programmer 	hugo
tested by	tobias

TC_S delivers the time it was last called on the output TC in seconds.

(*@KEY@:END_DESCRIPTION*)
FUNCTION_BLOCK TC_S

(*Group:Default*)

VAR_OUTPUT
	TC :	REAL;
END_VAR

VAR
	init :	BOOL;
	tx :	UDINT;
	last :	UDINT;
	T_PLC_US :	T_PLC_US;
END_VAR

(*@KEY@: WORKSHEET
NAME: TC_S
IEC_LANGUAGE: ST
*)
(* read system time and prepare input data *)
T_PLC_US();
tx:= T_PLC_US.T_PLC_US;

IF NOT init THEN
	init := TRUE;
	TC := 0.0;
ELSE
	tc := UDINT_TO_REAL(tx - last) * 1.0E-6;
END_IF;
last := tx;

(* revision history
hm	13. mar. 2008	rev 1.0
	original version

hm	16. mar 2008	rev 1.1
	added type conversion to avoid warnings under codesys 3.0

hm	11. mar. 2009	rev 1.2
	changed real constants to use dot syntax

*)

(*@KEY@: END_WORKSHEET *)
END_FUNCTION_BLOCK

(* ---- TC_US.ST ---- *)
(*@PROPERTIES_EX@
TYPE: POU
LOCALE: 0
IEC_LANGUAGE: ST
PLC_TYPE: independent
PROC_TYPE: independent
GROUP: ENGINEERING.MEASUREMENTS
*)
(*@KEY@:DESCRIPTION*)
version 1.0	13 mar 2008
programmer 	hugo
tested by	tobias

TC_US delivers the time it was last called on the output TC in Microseconds.
(*@KEY@:END_DESCRIPTION*)
FUNCTION_BLOCK TC_US

(*Group:Default*)

VAR_OUTPUT
	TC :	DWORD;
END_VAR

VAR
	init :	BOOL;
	tx :	UDINT;
	last :	UDINT;
	T_PLC_US :	T_PLC_US;
END_VAR

(*@KEY@: WORKSHEET
NAME: TC_US
IEC_LANGUAGE: ST
*)
(* read system time and prepare input data *)
T_PLC_US();
tx:= T_PLC_US.T_PLC_US;

IF NOT init THEN
	init := TRUE;
	TC := DWORD#0;
ELSE
	tc := UDINT_TO_DWORD(tx - last);
END_IF;
last := tx;

(* revision history
hm		13. mar. 2008	rev 1.0
	original version

*)
(*@KEY@: END_WORKSHEET *)
END_FUNCTION_BLOCK

(* ---- TEMPERATURE.ST ---- *)
(*@PROPERTIES_EX@
TYPE: POU
LOCALE: 0
IEC_LANGUAGE: ST
PLC_TYPE: independent
PROC_TYPE: independent
GROUP: ENGINEERING.CONVERSION
*)
(*@KEY@:DESCRIPTION*)
version 1.0	21 feb 2008
programmer 	hugo
tested by	oscat

this function converts different temperature units
any unused input can simply be left open.
different inputs connected at the same time will be added up.
(*@KEY@:END_DESCRIPTION*)
FUNCTION_BLOCK TEMPERATURE

(*Group:Default*)

VAR_INPUT
	K :	REAL;
	C :	REAL := -273.15;
	F :	REAL := -459.67;
	RE :	REAL := -218.52;
	RA :	REAL := 0.0;
END_VAR

VAR_OUTPUT
	YK :	REAL;
	YC :	REAL;
	YF :	REAL;
	YRE :	REAL;
	YRA :	REAL;
END_VAR

(*@KEY@: WORKSHEET
NAME: TEMPERATURE
IEC_LANGUAGE: ST
*)
YK := K + (C + 273.15) + (F + 459.67) * 0.555555555555 + (Re * 1.25 + 273.15) + (Ra * 0.555555555555);
YC := YK -273.15;
YF := YK * 1.8 - 459.67;
YRe := (YK - 273.15) * 0.8;
YRa := YK * 1.8;

(* revision history
hm	21. feb. 2008	rev 1.0
	original version

*)
(*@KEY@: END_WORKSHEET *)
END_FUNCTION_BLOCK

(* ---- TICKER.ST ---- *)
(*@PROPERTIES_EX@
TYPE: POU
LOCALE: 0
IEC_LANGUAGE: ST
PLC_TYPE: independent
PROC_TYPE: independent
GROUP: STRINGS
*)
(*@KEY@:DESCRIPTION*)
version 1.2	29. mar. 2008
programmer 	hugo
tested by	tobias

Ticker sends a substring of text with length N every TD Milliseconds to generate a ticker.
(*@KEY@:END_DESCRIPTION*)
FUNCTION_BLOCK TICKER

(*Group:Default*)

VAR_INPUT
	N :	INT;
	PT :	TIME;
	TEXT :	STRING;
END_VAR

VAR_OUTPUT
	DISPLAY :	STRING;
END_VAR

VAR
	delay :	TP;
	rollout :	STRING;
	text_len :	INT;
	rollout_step :	INT;
	step :	INT;
END_VAR

(*@KEY@: WORKSHEET
NAME: TICKER
IEC_LANGUAGE: ST
*)
(* generate next ticker when delay is low *)
text_len := LEN(text);

IF N < text_len THEN
	IF NOT delay.Q THEN

		IF step > text_len THEN
            rollout_step := 0;
            rollout := '';
            step := 0;
        END_IF;

        IF step + N > text_len THEN
		    (* increase step for next tick *)
		    step := step + 1;
            rollout_step := rollout_step +1;
		    (* extract dispay from text *)
		    display := MID(text, N - rollout_step, step);
            rollout := CONCAT(rollout,'#');
            display := CONCAT(display,rollout);
        ELSE
		    (* increase step for next tick *)
		    step := step + 1;
		    (* extract dispay from text *)
		    display := MID(text, N, step);
        END_IF;

		(* set delay timer for next tick *)
		delay(in := TRUE, PT := PT);
	ELSE;
		(* execute delay timer *)
		delay(in := FALSE);
	END_IF;
ELSE
	display := text;
END_IF;

(* revision history
hm	4. dec. 2007	rev 1.0
	original version

hm	15. dec. 2007	rev 1.1
	step now starts at 1 instaed of 0

hm	29. mar. 2008	rev 1.2
	changed STRING to STRING(STRING_LENGTH)
*)
(*@KEY@: END_WORKSHEET *)
END_FUNCTION_BLOCK

(* ---- TMAX.ST ---- *)
(*@PROPERTIES_EX@
TYPE: POU
LOCALE: 0
IEC_LANGUAGE: ST
PLC_TYPE: independent
PROC_TYPE: independent
GROUP: LOGIC.GENERATORS
*)
(*@KEY@:DESCRIPTION*)
version 1.0	20. jul. 2008
programmer 	hugo
tested by	oscat

Q of tmax will follow IN except that it forces a maximum ontime for the output Q.
the output Z will be active for one cycle if the output is forced low by the timeout.
(*@KEY@:END_DESCRIPTION*)
FUNCTION_BLOCK TMAX

(*Group:Default*)

VAR_INPUT
	IN :	BOOL;
	PT :	TIME;
END_VAR

VAR_OUTPUT
	Q :	BOOL;
	Z :	BOOL;
END_VAR

VAR
	tx :	TIME;
	start :	TIME;
	last_in :	BOOL;
	T_PLC_MS :	T_PLC_MS;
END_VAR

(*@KEY@: WORKSHEET
NAME: TMAX
IEC_LANGUAGE: ST
*)
(* read system timer *)
T_PLC_MS();
tx:= UDINT_TO_TIME(T_PLC_MS.T_PLC_MS);

Z := FALSE;

IF NOT in THEN
	Q := FALSE;
ELSIF IN AND NOT last_in THEN
	Q := TRUE;
	start := tx;
ELSIF (tx - start >= PT) AND Q THEN
	Q := FALSE;
	Z := TRUE;
END_IF;

last_in := IN;

(* revision history
hm	20. jul. 2008	rev 1.0
	original version

*)
(*@KEY@: END_WORKSHEET *)
END_FUNCTION_BLOCK

(* ---- TMIN.ST ---- *)
(*@PROPERTIES_EX@
TYPE: POU
LOCALE: 0
IEC_LANGUAGE: ST
PLC_TYPE: independent
PROC_TYPE: independent
GROUP: LOGIC.GENERATORS
*)
(*@KEY@:DESCRIPTION*)
version 1.0	21. jul. 2008
programmer 	hugo
tested by	oscat

Q of tMIN will follow IN except that it forces a minimum ontime for the output Q.
(*@KEY@:END_DESCRIPTION*)
FUNCTION_BLOCK TMIN

(*Group:Default*)

VAR_INPUT
	IN :	BOOL;
	PT :	TIME;
END_VAR

VAR_OUTPUT
	Q :	BOOL;
END_VAR

VAR
	pm :	TP;
END_VAR

(*@KEY@: WORKSHEET
NAME: TMIN
IEC_LANGUAGE: ST
*)
pm(in := IN, PT := PT);
Q := IN OR pm.Q;

(* revision history
hm	21. jul. 2008	rev 1.0
	original version

*)
(*@KEY@: END_WORKSHEET *)
END_FUNCTION_BLOCK

(* ---- TO_UML.ST ---- *)
(*@PROPERTIES_EX@
TYPE: POU
LOCALE: 0
IEC_LANGUAGE: ST
PLC_TYPE: independent
PROC_TYPE: independent
GROUP: STRINGS
*)
(*@KEY@:DESCRIPTION*)
version 1.1	17. dec. 2008
programmer 		hugo
tested by		tobias

to_uml converts a character above 127 to a two digit character below 127.
the character Ä is converted to Ae
(*@KEY@:END_DESCRIPTION*)
FUNCTION_BLOCK TO_UML

(*Group:Default*)

VAR_INPUT
	IN :	BYTE;
END_VAR

VAR_OUTPUT
	TO_UML :	STRING;
END_VAR

(*@KEY@: WORKSHEET
NAME: TO_UML
IEC_LANGUAGE: ST
*)
CASE _BYTE_TO_INT(in) OF
	196:	(* Ä *)
		TO_UML := 'Ae';
	214:	(* Ö *)
		TO_UML := 'Oe';
	220:	(* Ü *)
		TO_UML := 'Ue';
	223:	(* ß *)
		TO_UML := 'ss';
	228:	(* ä *)
		TO_UML := 'ae';
	246:	(* ö *)
		TO_UML := 'oe';
	252:	(* ü *)
		TO_UML := 'ue';
ELSE
	TO_UML := BYTE_TO_STRING(IN,'%c');
END_CASE;

(* revision history
hm	29. mar. 2008	rev 1.0
	original version

hm	17. dec. 2008	rev 1.1
	changes name of function chr to chr_to_string

*)
(*@KEY@: END_WORKSHEET *)
END_FUNCTION_BLOCK

(* ---- TOD_TO_STRING.ST ---- *)
(*@PROPERTIES_EX@
TYPE: POU
LOCALE: 0
IEC_LANGUAGE: ST
PLC_TYPE: independent
PROC_TYPE: independent
GROUP: EMULATION
*)
(*@KEY@:DESCRIPTION*)

(*@KEY@:END_DESCRIPTION*)
FUNCTION_BLOCK TOD_TO_STRING

(*Group:Default*)

VAR_INPUT
	ITOD :	UDINT;
END_VAR

VAR_OUTPUT
	TOD_STRING :	STRING;
END_VAR

VAR
	st_tmp1 :	STRING;
	st_tmp2 :	STRING;
	cur_hours :	INT;
END_VAR

(*@KEY@: WORKSHEET
NAME: TOD_TO_STRING
IEC_LANGUAGE: ST
*)
cur_hours := hour(ITOD);
IF cur_hours = 0 THEN
  st_tmp2 := '%01dh';
ELSE
  st_tmp2 := '%dh';
END_IF;

st_tmp1 := CONCAT(INT_TO_STRING(cur_hours,st_tmp2),INT_TO_STRING(minute(ITOD),'%02dm'));
TOD_STRING := CONCAT(st_tmp1,UDINT_TO_STRING(ITOD MOD UDINT#60000 / UDINT#1000,'%02us'));
(*@KEY@: END_WORKSHEET *)
END_FUNCTION_BLOCK

(* ---- TOF_1.ST ---- *)
(*@PROPERTIES_EX@
TYPE: POU
LOCALE: 0
IEC_LANGUAGE: ST
PLC_TYPE: independent
PROC_TYPE: independent
GROUP: LOGIC.GENERATORS
*)
(*@KEY@:DESCRIPTION*)
version 1.0	17. jul. 2008
programmer 	hugo
tested by	oscat

TOF_1 will extend a pulse on input in for PT seconds.
in addition the timer can be cleared asynchronously with rst.
TOF_1 is the same function as TOF from the standard LIB except the asynchronous reset input.
(*@KEY@:END_DESCRIPTION*)
FUNCTION_BLOCK TOF_1

(*Group:Default*)

VAR_INPUT
	IN :	BOOL;
	PT :	TIME;
	RST :	BOOL;
END_VAR

VAR_OUTPUT
	Q :	BOOL;
END_VAR

VAR
	start :	TIME;
	tx :	TIME;
	T_PLC_MS :	T_PLC_MS;
END_VAR

(*@KEY@: WORKSHEET
NAME: TOF_1
IEC_LANGUAGE: ST
*)
(* read system timer *)
T_PLC_MS();
tx:= UDINT_TO_TIME(T_PLC_MS.T_PLC_MS);

IF RST THEN
	Q := FALSE;
ELSIF IN THEN
	Q := TRUE;
	start := tx;
ELSIF tx - start >= PT THEN
	Q := FALSE;
END_IF;

(* revision history
hm	17. jul. 2008	rev 1.0
	original version

*)
(*@KEY@: END_WORKSHEET *)
END_FUNCTION_BLOCK

(* ---- TOGGLE.ST ---- *)
(*@PROPERTIES_EX@
TYPE: POU
LOCALE: 0
IEC_LANGUAGE: ST
PLC_TYPE: independent
PROC_TYPE: independent
GROUP: LOGIC.FF_EDGE_TRIGGERED
*)
(*@KEY@:DESCRIPTION*)
version 1.1	30. oct. 2008
programmer 	hugo
tested by	oscat

toggle flip flop the output changes state with every rising edge of clk.
(*@KEY@:END_DESCRIPTION*)
FUNCTION_BLOCK TOGGLE

(*Group:Default*)

VAR_INPUT
	CLK :	BOOL;
	RST :	BOOL;
END_VAR

VAR_OUTPUT
	Q :	BOOL;
END_VAR

VAR
	edge :	BOOL;
END_VAR

(*@KEY@: WORKSHEET
NAME: TOGGLE
IEC_LANGUAGE: ST
*)
IF rst THEN
	Q := FALSE;
ELSIF clk AND NOT edge THEN
	Q := NOT Q;
END_IF;
edge := clk;

(* revision history

hm	13.9.2007		rev 1.0
	original version

hm	30. oct. 2008	rev 1.1
	deleted unnecessary init

*)
(*@KEY@: END_WORKSHEET *)
END_FUNCTION_BLOCK

(* ---- TONOF.ST ---- *)
(*@PROPERTIES_EX@
TYPE: POU
LOCALE: 0
IEC_LANGUAGE: ST
PLC_TYPE: independent
PROC_TYPE: independent
GROUP: LOGIC.GENERATORS
*)
(*@KEY@:DESCRIPTION*)
version 1.2	21. jul 2009
programmer 	hugo
tested by	tobias

TONOF generated a TON and TOF Delay for the Input N TON (T1) and TOF (T2) can be configured separately

(*@KEY@:END_DESCRIPTION*)
FUNCTION_BLOCK TONOF

(*Group:Default*)

VAR_INPUT
	IN :	BOOL;
	T_ON :	TIME;
	T_OFF :	TIME;
END_VAR

VAR_OUTPUT
	Q :	BOOL;
END_VAR

VAR
	X :	TON;
	old :	BOOL;
	mode :	BOOL;
END_VAR

(*@KEY@: WORKSHEET
NAME: TONOF
IEC_LANGUAGE: ST
*)
IF IN XOR old THEN
  X(IN := FALSE, PT := SEL_TIME(IN,T_OFF,T_ON));
  mode := IN;
  old := IN;
END_IF;
X(IN := TRUE);
IF X.Q THEN Q := mode;END_IF;

(* revision history
hm	10. dec 2007	rev 1.0
	original version

hm	17. sep. 2007	rev 1.1
	improved performance

hm	21. jul. 2009	rev 1.2
	fixed a timing probelm

*)

(*@KEY@: END_WORKSHEET *)
END_FUNCTION_BLOCK

(* ---- TP_1.ST ---- *)
(*@PROPERTIES_EX@
TYPE: POU
LOCALE: 0
IEC_LANGUAGE: ST
PLC_TYPE: independent
PROC_TYPE: independent
GROUP: LOGIC.GENERATORS
*)
(*@KEY@:DESCRIPTION*)
version 1.0	28. jun. 2008
programmer 	hugo
tested by	oscat

TP_1 generates a pulse every time it is calles with in := TRUE.
in addition the timer can be cleared asynchronously with rst.
the timer can be retriggered as often as necessary. it will count PT from the last trigger.
(*@KEY@:END_DESCRIPTION*)
FUNCTION_BLOCK TP_1

(*Group:Default*)

VAR_INPUT
	IN :	BOOL;
	PT :	TIME;
	RST :	BOOL;
END_VAR

VAR_OUTPUT
	Q :	BOOL;
END_VAR

VAR
	tx :	TIME;
	start :	TIME;
	ix :	BOOL;
	T_PLC_MS :	T_PLC_MS;
END_VAR

(*@KEY@: WORKSHEET
NAME: TP_1
IEC_LANGUAGE: ST
*)
(* read system timer *)
(* read system_time *)
T_PLC_MS();
tx := UDINT_TO_TIME(T_PLC_MS.T_PLC_MS);

IF RST THEN
	Q := FALSE;
ELSIF IN AND NOT ix THEN
	Q := TRUE;
	start := tx;
ELSIF tx - start >= PT THEN
	Q := FALSE;
END_IF;

ix:= IN;

(* revision history
hm	28. jun. 2008
	original version

*)
(*@KEY@: END_WORKSHEET *)
END_FUNCTION_BLOCK

(* ---- TP_1D.ST ---- *)
(*@PROPERTIES_EX@
TYPE: POU
LOCALE: 0
IEC_LANGUAGE: ST
PLC_TYPE: independent
PROC_TYPE: independent
GROUP: LOGIC.GENERATORS
*)
(*@KEY@:DESCRIPTION*)
version 1.0	28. jun. 2008
programmer 	hugo
tested by	oscat

TP_2 generates a pulse every time it is calles with in := TRUE.
the module will reset IN by itself so no clearing of in is necessary.
in addition the timer can be cleared asynchronously with rst.
also the rst input is cleared by the module itself.
the timer can be retriggered as often as necessary. it will count PT from the last trigger.
after the time PT1 is elapsed, the timer blocks itself for PT2 and only allow new sequences after PT2 has elapsed.
(*@KEY@:END_DESCRIPTION*)
FUNCTION_BLOCK TP_1D

(*Group:Default*)

VAR_INPUT
	IN :	BOOL;
	PT1 :	TIME;
	PTD :	TIME;
	RST :	BOOL;
END_VAR

VAR_OUTPUT
	Q :	BOOL;
	W :	BOOL;
END_VAR

VAR
	tx :	TIME;
	start :	TIME;
	ix :	BOOL;
	T_PLC_MS :	T_PLC_MS;
END_VAR

(*@KEY@: WORKSHEET
NAME: TP_1D
IEC_LANGUAGE: ST
*)
(* read system_time *)
T_PLC_MS();
tx := UDINT_TO_TIME(T_PLC_MS.T_PLC_MS);

IF RST THEN
	Q := FALSE;
	rst := FALSE;
	W := FALSE;
ELSIF W THEN
	IF tx - start >= PTD THEN
		W := FALSE;
	END_IF;
ELSIF IN AND NOT ix THEN
	Q := TRUE;
	start := tx;
	in := FALSE;
ELSIF tx - start >= PT1 THEN
	Q := FALSE;
	W := TRUE;
	start := tx;
END_IF;

ix := IN;

(* revision history
hm	28. jun. 2008
	original version

*)
(*@KEY@: END_WORKSHEET *)
END_FUNCTION_BLOCK

(* ---- TP_X.ST ---- *)
(*@PROPERTIES_EX@
TYPE: POU
LOCALE: 0
IEC_LANGUAGE: ST
PLC_TYPE: independent
PROC_TYPE: independent
GROUP: LOGIC.GENERATORS
*)
(*@KEY@:DESCRIPTION*)
version 1.3	17. dec. 2008
programmer 	hugo
tested by	oscat

retriggerable edge triggered pulse similar to TP but with a retrigger function
if the pt input is 0 then output is always low.
(*@KEY@:END_DESCRIPTION*)
FUNCTION_BLOCK TP_X

(*Group:Default*)

VAR_INPUT
	IN :	BOOL;
	PT :	TIME;
END_VAR

VAR_OUTPUT
	Q :	BOOL;
	ET :	TIME;
END_VAR

VAR
	edge :	BOOL;
	start :	TIME;
	tx :	TIME;
	T_PLC_MS :	T_PLC_MS;
END_VAR

(*@KEY@: WORKSHEET
NAME: TP_X
IEC_LANGUAGE: ST
*)
(* read system_time *)
T_PLC_MS();
tx := UDINT_TO_TIME(T_PLC_MS.T_PLC_MS);

(* rising edge trigger *)
IF IN AND NOT edge THEN
	start := tx;
	Q := PT > t#0ms;
ELSIF Q THEN
	ET := tx - start;
	IF ET >= PT THEN
		Q := FALSE;
		ET := t#0ms;
	END_IF;
END_IF;
edge := IN;

(* revision history
hm	4. aug 2006		rev 1.0
	original version

hm	17. sep 2007	rev 1.1
	replaced time() with T_PLC_MS() for compatibility reasons

hm	19. oct. 2008	rev 1.2
	renamed to TP_R to TP_X for compatibility reasons

hm	17. dec. 2008	rev 1.3
	code optimized

*)
(*@KEY@: END_WORKSHEET *)
END_FUNCTION_BLOCK

(* ---- TREND.ST ---- *)
(*@PROPERTIES_EX@
TYPE: POU
LOCALE: 0
IEC_LANGUAGE: ST
PLC_TYPE: independent
PROC_TYPE: independent
GROUP: ENGINEERING.SIGNAL_PROCESSING
*)
(*@KEY@:DESCRIPTION*)
version 1.0	21. aug. 2009
programmer 	hugo
tested by	oscat

trend analyses the trend of a input signal.
The Output Q is True if the input X is >= last_X and is false if the input X is <= last_X
in addition to the trend the output TU will be high for one cycle to signal a rising of the input value X
and  TD will signal a decreasing value on the input X.
in case of a change the output D will show the delta of the input to the last input value.

(*@KEY@:END_DESCRIPTION*)
FUNCTION_BLOCK TREND

(*Group:Default*)

VAR_INPUT
	X :	REAL;
END_VAR

VAR_OUTPUT
	Q :	BOOL;
	TU :	BOOL;
	TD :	BOOL;
	D :	REAL;
END_VAR

VAR
	last_x :	REAL;
END_VAR

(*@KEY@: WORKSHEET
NAME: TREND
IEC_LANGUAGE: ST
*)
TU := X > last_X;
TD := X < last_X;
Q := TU OR TD;
D := X - LAST_X;

last_X := X;

(* revision history
hm	21. aug. 2009	rev 1.0
	original version

*)

(*@KEY@: END_WORKSHEET *)
END_FUNCTION_BLOCK

(* ---- TREND_DW.ST ---- *)
(*@PROPERTIES_EX@
TYPE: POU
LOCALE: 0
IEC_LANGUAGE: ST
PLC_TYPE: independent
PROC_TYPE: independent
GROUP: ENGINEERING.SIGNAL_PROCESSING
*)
(*@KEY@:DESCRIPTION*)
version 1.2	14. mar. 2009
programmer 	hugo
tested by	oscat

trend_DW analyses the trend of a input signal.
The Output Q is True if the input X is >= last_X and is false if the input X is <= last_X
in addition to the trend the output TU will be high for one cycle to signal a rising of the input value X
and  TD will signal a decreasing value on the input X.
in case of a change the output D will show the delta of the input to the last input value.

(*@KEY@:END_DESCRIPTION*)
FUNCTION_BLOCK TREND_DW

(*Group:Default*)

VAR_INPUT
	X :	DWORD;
END_VAR

VAR_OUTPUT
	Q :	BOOL;
	TU :	BOOL;
	TD :	BOOL;
	D :	DWORD;
END_VAR

VAR
	LAST_X :	DWORD;
END_VAR

(*@KEY@: WORKSHEET
NAME: TREND_DW
IEC_LANGUAGE: ST
*)
IF X > last_X THEN
	TU := TRUE;
	TD := FALSE;
	D := UDINT_TO_DWORD(DWORD_TO_UDINT(X) - DWORD_TO_UDINT(last_X));
	Q := TRUE;
ELSIF X < last_X THEN
	TD := TRUE;
	TU := FALSE;
	D := UDINT_TO_DWORD(DWORD_TO_UDINT(last_X) - DWORD_TO_UDINT(X));
	Q := FALSE;
ELSE
	TU := FALSE;
	TD := FALSE;
	D := DWORD#0;
END_IF;
last_X := X;

(* revision history
hm	21. nov. 2008	rev 1.0
	original version

hm	20. feb. 2009	rev 1.1
	added outputs TU, TD and D

hm	14. mar. 2009	rev 1.2
	removed double assignments

*)

(*@KEY@: END_WORKSHEET *)
END_FUNCTION_BLOCK

(* ---- TRIM.ST ---- *)
(*@PROPERTIES_EX@
TYPE: POU
LOCALE: 0
IEC_LANGUAGE: ST
PLC_TYPE: independent
PROC_TYPE: independent
GROUP: STRINGS
*)
(*@KEY@:DESCRIPTION*)
version 1.2	29. mar. 2008
programmer 	hugo
tested by	tobias

the function deletes all blanks within a string.
(*@KEY@:END_DESCRIPTION*)
FUNCTION_BLOCK TRIM

(*Group:Default*)

VAR_INPUT
	STR :	STRING;
END_VAR

VAR_OUTPUT
	TRIM :	STRING;
END_VAR

VAR
	pos :	INT;
END_VAR

(*@KEY@: WORKSHEET
NAME: TRIM
IEC_LANGUAGE: ST
*)
trim := str;
REPEAT
	pos := FIND(trim,' ');
	IF pos > 0 THEN trim := REPLACE(trim,'',1,pos); END_IF;
UNTIL pos = 0 END_REPEAT;

(* revision histroy
hm	6.10.2006		rev 1.0
	original release

hm	20. mar. 2008	rev 1.1
	avoid to call replace with pos = 0 because some systems will produce an error

hm	29. mar. 2008	rev 1.2
	changed STRING to STRING(STRING_LENGTH)
*)
(*@KEY@: END_WORKSHEET *)
END_FUNCTION_BLOCK

(* ---- TRIM1.ST ---- *)
(*@PROPERTIES_EX@
TYPE: POU
LOCALE: 0
IEC_LANGUAGE: ST
PLC_TYPE: independent
PROC_TYPE: independent
GROUP: STRINGS
*)
(*@KEY@:DESCRIPTION*)
version 1.2	29. mar. 2008
programmer 	hugo
tested by	tobias

the function replaces all multiple blanks within a string by only one blank.
leading and ending blanks will be deleted
(*@KEY@:END_DESCRIPTION*)
FUNCTION_BLOCK TRIM1

(*Group:Default*)

VAR_INPUT
	STR :	STRING;
END_VAR

VAR_OUTPUT
	TRIM1 :	STRING;
END_VAR

VAR
	pos :	INT;
	st_temp :	STRING;
END_VAR

(*@KEY@: WORKSHEET
NAME: TRIM1
IEC_LANGUAGE: ST
*)
trim1 := str;
REPEAT
	pos := FIND(trim1,'  ');
	IF pos > 0 THEN
	  st_temp := trim1;
	  trim1 := REPLACE(trim1,' ',2,pos);
    END_IF;
UNTIL pos = 0 END_REPEAT;
(* beginning and ending blanks need to be stripped off *)
st_temp := LEFT(trim1,1);
IF EQ_STRING(st_temp,' ') THEN trim1 := DELETE(trim1,1,1); END_IF;
st_temp := RIGHT(trim1,1);
IF EQ_STRING(st_temp,' ') THEN trim1 := DELETE(trim1,1,LEN(trim1)); END_IF;

(* revision histroy
hm	4. feb. 2008    rev 1.0
	original release

hm	20. mar. 2008	rev 1.1
	avoid to call replace with pos = 0 because some systems will produce an error

hm	29. mar. 2008	rev 1.2
	changed STRING to STRING(STRING_LENGTH)
*)
(*@KEY@: END_WORKSHEET *)
END_FUNCTION_BLOCK

(* ---- TRIME.ST ---- *)
(*@PROPERTIES_EX@
TYPE: POU
LOCALE: 0
IEC_LANGUAGE: ST
PLC_TYPE: independent
PROC_TYPE: independent
GROUP: STRINGS
*)
(*@KEY@:DESCRIPTION*)
version 1.0	28. mar. 2008
programmer 	hugo
tested by	tobias

this function deletes all leading and ending blanks of a string.
(*@KEY@:END_DESCRIPTION*)
FUNCTION_BLOCK TRIME

(*Group:Default*)

VAR_INPUT
	STR :	STRING;
END_VAR

VAR_OUTPUT
	TRIME :	STRING;
END_VAR

(*@KEY@: WORKSHEET
NAME: TRIME
IEC_LANGUAGE: ST
*)
TRIME := str;
IF LEN(TRIME) < 1 THEN RETURN; END_IF;

WHILE (GET_CHAR(TRIME,1) = 32) DO
	TRIME := DELETE(TRIME,1,1);
END_WHILE;

(* ending blanks need to be stripped off *)
WHILE (GET_CHAR(TRIME,LEN(TRIME)) = 32) DO
	TRIME := DELETE(TRIME,1,LEN(TRIME));
END_WHILE;

(* revision histroy
hm		4. feb. 2008		rev 1.0
	original release

*)
(*@KEY@: END_WORKSHEET *)
END_FUNCTION_BLOCK

(* ---- TUNE.ST ---- *)
(*@PROPERTIES_EX@
TYPE: POU
LOCALE: 0
IEC_LANGUAGE: ST
PLC_TYPE: independent
PROC_TYPE: independent
GROUP: ENGINEERING.AUTOMATION
*)
(*@KEY@:DESCRIPTION*)
version 1.2	11. mar. 2009
programmer 	hugo
tested by	tobias

tune generates an output signal which is set by input switches.
up to 4 switsches can be used to tune the signal up or down.

(*@KEY@:END_DESCRIPTION*)
FUNCTION_BLOCK TUNE

(*Group:Default*)

VAR_INPUT
	SET :	BOOL;
	SU :	BOOL;
	SD :	BOOL;
	RST :	BOOL;
	SS :	REAL := 0.1;
	LIMIT_L :	REAL;
	LIMIT_H :	REAL := 100.0;
	RST_VAL :	REAL;
	SET_VAL :	REAL := 100.0;
	T1 :	TIME := T#500ms;
	T2 :	TIME := T#2s;
	S1 :	REAL := 2.0;
	S2 :	REAL := 10.0;
END_VAR

VAR_OUTPUT
	Y :	REAL;
END_VAR

VAR
	tx :	UDINT;
	start :	UDINT;
	start2 :	UDINT;
	state :	INT;
	in :	BOOL;
	step :	REAL;
	speed :	REAL;
	Y_start :	REAL;
	Y_start2 :	REAL;
	T_PLC_MS :	T_PLC_MS;
END_VAR

(*@KEY@: WORKSHEET
NAME: TUNE
IEC_LANGUAGE: ST
*)
(* read system_time *)
T_PLC_MS();
tx:= T_PLC_MS.T_PLC_MS;

IF rst THEN
	Y := RST_val;
	state := 0;
ELSIF set THEN
	Y := SET_val;
	state := 0;
ELSIF state > 0 THEN
	(* key has been pushed state machine operating *)
	(* first read the correct input *)
	IF state = 1 THEN
		(* step up *)
		in := su;
	ELSE
		(* step down *)
		in := sd;
	END_IF;
	(* check for single step operation *)
	IF NOT in AND tx - start <= TIME_TO_UDINT(T1) THEN
		Y := Y_start + step;
		state := 0;
	(* check if fast ramp needs to be generated *)
	ELSIF in AND tx - start >= TIME_TO_UDINT(T2) THEN
		Y := Y_start2 + UDINT_TO_REAL(tx - start2) * s2 / speed;
	(* check if slow ramp needs to be generated *)
	ELSIF in AND tx - start >= TIME_TO_UDINT(T1) THEN
		Y := Y_start + UDINT_TO_REAL(tx - start - TIME_TO_UDINT(T1)) * S1 / speed;
		start2 := tx;
		Y_start2 := Y;
	ELSIF NOT in THEN
		state := 0;
	END_IF;
ELSIF su THEN
	(* slow step up *)
	state := 1;
	start := tx;
	step := ss;
	speed := 1000.0;
	Y_start := Y;
ELSIF sd THEN
	(* slow step down *)
	state := 2;
	start := tx;
	step := -ss;
	speed := -1000.0;
	Y_start := Y;
END_IF;

(* make sure output does not exceed limits *)
Y := LIMIT(LIMIT_L, Y, LIMIT_H);

(* revision history
hm	3.11.2007		rev 1.0
	original version

hm	16. mar. 2008	rev 1.1
	added type conversions to avoid warnings under codesys 3.0

hm	11. mar. 2009	rev 1.2
	real constants updated to new systax using dot

*)
(*@KEY@: END_WORKSHEET *)
END_FUNCTION_BLOCK

(* ---- TUNE2.ST ---- *)
(*@PROPERTIES_EX@
TYPE: POU
LOCALE: 0
IEC_LANGUAGE: ST
PLC_TYPE: independent
PROC_TYPE: independent
GROUP: ENGINEERING.AUTOMATION
*)
(*@KEY@:DESCRIPTION*)
version 1.2	11. mar. 2009
programmer 	hugo
tested by	tobias

tune2 generates an output signal which is set by input switches.
up to 4 switsches can be used to tune the signal up or down.

(*@KEY@:END_DESCRIPTION*)
FUNCTION_BLOCK TUNE2

(*Group:Default*)

VAR_INPUT
	SET :	BOOL;
	SU :	BOOL;
	SD :	BOOL;
	FU :	BOOL;
	FD :	BOOL;
	RST :	BOOL;
	SS :	REAL := 0.1;
	FS :	REAL := 5.0;
	LIMIT_L :	REAL;
	LIMIT_H :	REAL := 100.0;
	RST_VAL :	REAL;
	SET_VAL :	REAL := 100.0;
	TR :	TIME := T#500ms;
	S1 :	REAL := 2.0;
	S2 :	REAL := 10.0;
END_VAR

VAR_OUTPUT
	Y :	REAL;
END_VAR

VAR
	tx :	UDINT;
	start :	UDINT;
	state :	INT;
	in :	BOOL;
	step :	REAL;
	speed :	REAL;
	Y_start :	REAL;
	T_PLC_MS :	T_PLC_MS;
END_VAR

(*@KEY@: WORKSHEET
NAME: TUNE2
IEC_LANGUAGE: ST
*)
(* read system time *)
T_PLC_MS();
tx:= T_PLC_MS.T_PLC_MS;

IF rst THEN
	Y := RST_val;
	state := 0;
ELSIF set THEN
	Y := SET_val;
	state := 0;
ELSIF state > 0 THEN
	(* key has been pushed state machine operating *)
	(* first read the correct input *)
	CASE state OF
		1 :	(* slow up *)
			in := su;
		2 :	(* slow down *)
			in := sd;
		3 :	(* fast up *)
			in := fu;
		4 :	(* fast down *)
			in := fd;
	END_CASE;
	(* check for single step operation *)
	IF NOT in AND tx - start <= TIME_TO_UDINT(TR) THEN
		Y := Y_start + step;
		state := 0;
	(* check if ramp needs to be generated *)
	ELSIF in AND tx - start >= TIME_TO_UDINT(TR) THEN
		Y := Y_start + UDINT_TO_REAL(tx - start - TIME_TO_UDINT(TR)) * speed;
	ELSIF NOT in THEN
		state := 0;
	END_IF;
ELSIF su THEN
	(* slow step up *)
	state := 1;
	start := tx;
	step := ss;
	speed := s1 * 1.0E-3;
	Y_start := Y;
ELSIF sd THEN
	(* slow step down *)
	state := 2;
	start := tx;
	step := -ss;
	speed := -s1 * 1.0E-3;
	Y_start := Y;
ELSIF fu THEN
	(* fast step up *)
	state := 3;
	start := tx;
	step := fs;
	speed := s2 * 1.0E-3;
	y_start := Y;
ELSIF fd THEN
	(* fast step down *)
	state := 4;
	start := tx;
	step := -fs;
	speed := -s2 * 1.0E-3;
	y_start := Y;
END_IF;

(* make sure output does not exceed limits *)
Y := LIMIT(LIMIT_L, Y, LIMIT_H);

(* revision history
hm	3.11.2007		rev 1.0
	original version

hm	16. 3. 2008	rev 1.1
	added type conversions to avoid warnings in codesys 3.0
	improved performance

hm	11. mar. 2009	rev 1.2
	real constants updated to new systax using dot

*)
(*@KEY@: END_WORKSHEET *)
END_FUNCTION_BLOCK

(* ---- UPPERCASE.ST ---- *)
(*@PROPERTIES_EX@
TYPE: POU
LOCALE: 0
IEC_LANGUAGE: ST
PLC_TYPE: independent
PROC_TYPE: independent
GROUP: STRINGS
*)
(*@KEY@:DESCRIPTION*)
version 1.3	29. mar. 2008
programmer 	hugo
tested by	tobias

uppercase returns str while all letters a..z and ä,ö,ü are converted to uppercase
(*@KEY@:END_DESCRIPTION*)
FUNCTION_BLOCK UPPERCASE

(*Group:Default*)

VAR_INPUT
	STR :	STRING;
END_VAR

VAR_OUTPUT
	UPPERCASE :	STRING;
END_VAR

VAR
	char :	BYTE;
	char2 :	BYTE;
	pos :	INT;
	l :	INT;
	str_temp :	STRING;
END_VAR

(*@KEY@: WORKSHEET
NAME: UPPERCASE
IEC_LANGUAGE: ST
*)
UPPERCASE := str;
l := LEN(str);
FOR pos := 1 TO l DO
    char := INT_TO_BYTE(GET_CHAR(str,pos));
	char2 := TO_UPPER(char);
    IF char <> char2 THEN
    	str_temp := UPPERCASE;
      	UPPERCASE := REPLACE(str_temp,BYTE_TO_STRING(char2,'%c'),1,pos);
	END_IF;
END_FOR;

(* revision histroy
hm	6. oct. 2006	rev 1.0
	original release

hm	4. feb. 2008	rev 1.1
	improved performance
	added Ä,Ö,Ü

hm	6. mar. 2008	rev 1.2
	added support for exteded Ascii

hm	29. mar. 2008	rev 1.3
	changed STRING to STRING(STRING_LENGTH)
*)
(*@KEY@: END_WORKSHEET *)
END_FUNCTION_BLOCK

(* ---- V3_ABS.ST ---- *)
(*@PROPERTIES_EX@
TYPE: POU
LOCALE: 0
IEC_LANGUAGE: ST
PLC_TYPE: independent
PROC_TYPE: independent
GROUP: MATHEMATICAL.VEKTORMATHEMATIK
*)
(*@KEY@:DESCRIPTION*)
version 1.0	11 dec 2007
programmer 	hugo
tested by	tobias

this function calculates the length of a vectors in a 3 dimensional space
(*@KEY@:END_DESCRIPTION*)
FUNCTION_BLOCK V3_ABS

(*Group:Default*)

VAR_INPUT
	A :	oscat_vector_3;
END_VAR

VAR_OUTPUT
	V3_ABS :	REAL;
END_VAR

(*@KEY@: WORKSHEET
NAME: V3_ABS
IEC_LANGUAGE: ST
*)
V3_ABS := SQRT(A.X * A.X + A.Y * A.Y + A.Z * A.Z);

(* revision history
hm		11 dec 2007	rev 1.0
	original version

*)
(*@KEY@: END_WORKSHEET *)
END_FUNCTION_BLOCK

(* ---- V3_ADD.ST ---- *)
(*@PROPERTIES_EX@
TYPE: POU
LOCALE: 0
IEC_LANGUAGE: ST
PLC_TYPE: independent
PROC_TYPE: independent
GROUP: MATHEMATICAL.VEKTORMATHEMATIK
*)
(*@KEY@:DESCRIPTION*)
version 1.0	11 dec 2007
programmer 	hugo
tested by	tobias

this function adds two vectors in a 3 dimensional space
(*@KEY@:END_DESCRIPTION*)
FUNCTION_BLOCK V3_ADD

(*Group:Default*)

VAR_INPUT
	A :	oscat_vector_3;
	B :	oscat_vector_3;
END_VAR

VAR_OUTPUT
	V3_ADD :	oscat_vector_3;
END_VAR

(*@KEY@: WORKSHEET
NAME: V3_ADD
IEC_LANGUAGE: ST
*)
V3_ADD.X := A.X + B.X;
V3_ADD.Y := A.Y + B.Y;
V3_ADD.Z := A.Z + B.Z;

(* revision history
hm		11 dec 2007	rev 1.0
	original version

*)
(*@KEY@: END_WORKSHEET *)
END_FUNCTION_BLOCK

(* ---- V3_ANG.ST ---- *)
(*@PROPERTIES_EX@
TYPE: POU
LOCALE: 0
IEC_LANGUAGE: ST
PLC_TYPE: independent
PROC_TYPE: independent
GROUP: MATHEMATICAL.VEKTORMATHEMATIK
*)
(*@KEY@:DESCRIPTION*)
version 1.1	10. mar. 2009
programmer 	hugo
tested by	tobias

this function calculates the angle between two vectors in a 3 dimensional space

(*@KEY@:END_DESCRIPTION*)
FUNCTION_BLOCK V3_ANG

(*Group:Default*)

VAR_INPUT
	A :	oscat_vector_3;
	B :	oscat_vector_3;
END_VAR

VAR_OUTPUT
	V3_ANG :	REAL;
END_VAR

VAR
	d :	REAL;
	V3_ABS :	V3_ABS;
	V3_DPRO :	V3_DPRO;
END_VAR

(*@KEY@: WORKSHEET
NAME: V3_ANG
IEC_LANGUAGE: ST
*)

V3_ABS(A:=A);
d :=V3_ABS.V3_ABS;

V3_ABS(A:=B);
d := d * V3_ABS.V3_ABS;

IF d > 0.0 THEN
    V3_DPRO(A:=A,B:=B);
	V3_ANG := ACOS(LIMIT(-1.0, V3_DPRO.V3_DPRO / d,1.0));
ELSE
    V3_ANG := 0.0;

END_IF;

(* revision history
hm	11. dec. 2007	rev 1.0
	original version

hm	10. mar. 2009	rev 1.1
	changed syntax of real constants to 0.0

*)
(*@KEY@: END_WORKSHEET *)
END_FUNCTION_BLOCK

(* ---- V3_DPRO.ST ---- *)
(*@PROPERTIES_EX@
TYPE: POU
LOCALE: 0
IEC_LANGUAGE: ST
PLC_TYPE: independent
PROC_TYPE: independent
GROUP: MATHEMATICAL.VEKTORMATHEMATIK
*)
(*@KEY@:DESCRIPTION*)
version 1.0	11 dec 2007
programmer 	hugo
tested by	tobias

this function calculates the dot product of two vectors in 3 dimensional space
(*@KEY@:END_DESCRIPTION*)
FUNCTION_BLOCK V3_DPRO

(*Group:Default*)

VAR_INPUT
	A :	oscat_vector_3;
	B :	oscat_vector_3;
END_VAR

VAR_OUTPUT
	V3_DPRO :	REAL;
END_VAR

(*@KEY@: WORKSHEET
NAME: V3_DPRO
IEC_LANGUAGE: ST
*)
V3_DPRO := A.X * B.X + A.Y * B.Y + A.Z * B.Z;

(* revision history
hm		11 dec 2007	rev 1.0
	original version

*)
(*@KEY@: END_WORKSHEET *)
END_FUNCTION_BLOCK

(* ---- V3_NORM.ST ---- *)
(*@PROPERTIES_EX@
TYPE: POU
LOCALE: 0
IEC_LANGUAGE: ST
PLC_TYPE: independent
PROC_TYPE: independent
GROUP: MATHEMATICAL.VEKTORMATHEMATIK
*)
(*@KEY@:DESCRIPTION*)
version 1.1	10. mar. 2009
programmer 	hugo
tested by	tobias

this function generates a vectors with absolute length 1 from a vector A in a 3 dimensional space

(*@KEY@:END_DESCRIPTION*)
FUNCTION_BLOCK V3_NORM

(*Group:Default*)

VAR_INPUT
	A :	oscat_vector_3;
END_VAR

VAR_OUTPUT
	V3_NORM :	oscat_vector_3;
END_VAR

VAR
	la :	REAL;
	V3_SMUL :	V3_SMUL;
	V3_ABS :	V3_ABS;
END_VAR

(*@KEY@: WORKSHEET
NAME: V3_NORM
IEC_LANGUAGE: ST
*)

V3_ABS(A:=A);
la:=V3_ABS.V3_ABS;

IF la > 0.0 THEN
    V3_SMUL(A:=A,M:=1.0/la);
    V3_NORM:=V3_SMUL.V3_SMUL;
ELSE
    V3_NORM.X := 0.0;
    V3_NORM.Y := 0.0;
    V3_NORM.Z := 0.0;
END_IF;

(* revision history
hm	11 dec 2007	rev 1.0
	original version

hm	10. mar. 2009	rev 1.1
	changed syntax of real constants to 0.0

*)
(*@KEY@: END_WORKSHEET *)
END_FUNCTION_BLOCK

(* ---- V3_NUL.ST ---- *)
(*@PROPERTIES_EX@
TYPE: POU
LOCALE: 0
IEC_LANGUAGE: ST
PLC_TYPE: independent
PROC_TYPE: independent
GROUP: MATHEMATICAL.VEKTORMATHEMATIK
*)
(*@KEY@:DESCRIPTION*)
version 1.1	10. mar. 2009
programmer 	hugo
tested by	tobias

this function checks if a vectors in a null Vector
(*@KEY@:END_DESCRIPTION*)
FUNCTION_BLOCK V3_NUL

(*Group:Default*)

VAR_INPUT
	A :	oscat_vector_3;
END_VAR

VAR_OUTPUT
	V3_NUL :	BOOL;
END_VAR

(*@KEY@: WORKSHEET
NAME: V3_NUL
IEC_LANGUAGE: ST
*)
V3_NUL := A.X = 0.0 AND A.Y = 0.0 AND A.Z = 0.0;

(* revision history
hm	12 dec 2007	rev 1.0
	original version

hm	10. mar. 2009	rev 1.1
	changed syntax of real constants to 0.0

*)
(*@KEY@: END_WORKSHEET *)
END_FUNCTION_BLOCK

(* ---- V3_PAR.ST ---- *)
(*@PROPERTIES_EX@
TYPE: POU
LOCALE: 0
IEC_LANGUAGE: ST
PLC_TYPE: independent
PROC_TYPE: independent
GROUP: MATHEMATICAL.VEKTORMATHEMATIK
*)
(*@KEY@:DESCRIPTION*)
version 1.1	10. mar. 2009
programmer 	hugo
tested by	tobias

this function checks if two vectors in a 3 dimensional space are parallel.
which means the two vectors have the same direction
(*@KEY@:END_DESCRIPTION*)
FUNCTION_BLOCK V3_PAR

(*Group:Default*)

VAR_INPUT
	A :	oscat_vector_3;
	B :	oscat_vector_3;
END_VAR

VAR_OUTPUT
	V3_PAR :	BOOL;
END_VAR

VAR
	V3_XPRO :	V3_XPRO;
	V3_ABS :	V3_ABS;
END_VAR

(*@KEY@: WORKSHEET
NAME: V3_PAR
IEC_LANGUAGE: ST
*)
V3_XPRO(A:=A,B:=B);
V3_ABS(A:=V3_XPRO.V3_XPRO);

V3_PAR := V3_ABS.V3_ABS = 0.0;

(* revision history
hm	11 dec 2007	rev 1.0
	original version

hm	10. mar. 2009	rev 1.1
	changed syntax of real constants to 0.0

*)
(*@KEY@: END_WORKSHEET *)
END_FUNCTION_BLOCK

(* ---- V3_REV.ST ---- *)
(*@PROPERTIES_EX@
TYPE: POU
LOCALE: 0
IEC_LANGUAGE: ST
PLC_TYPE: independent
PROC_TYPE: independent
GROUP: MATHEMATICAL.VEKTORMATHEMATIK
*)
(*@KEY@:DESCRIPTION*)
version 1.0	11 dec 2007
programmer 	hugo
tested by	tobias

this function reverses a vector in a 3 dimensional space
(*@KEY@:END_DESCRIPTION*)
FUNCTION_BLOCK V3_REV

(*Group:Default*)

VAR_INPUT
	A :	oscat_vector_3;
END_VAR

VAR_OUTPUT
	V3_REV :	oscat_vector_3;
END_VAR

(*@KEY@: WORKSHEET
NAME: V3_REV
IEC_LANGUAGE: ST
*)
V3_REV.X := -A.X;
V3_REV.Y := -A.Y;
V3_REV.Z := -A.Z;

(* revision history
hm		11 dec 2007	rev 1.0
	original version

*)
(*@KEY@: END_WORKSHEET *)
END_FUNCTION_BLOCK

(* ---- V3_SMUL.ST ---- *)
(*@PROPERTIES_EX@
TYPE: POU
LOCALE: 0
IEC_LANGUAGE: ST
PLC_TYPE: independent
PROC_TYPE: independent
GROUP: MATHEMATICAL.VEKTORMATHEMATIK
*)
(*@KEY@:DESCRIPTION*)
version 1.0	11 dec 2007
programmer 	hugo
tested by	tobias

this function multiplies a vectors in a 3 dimensional space with a skalar M
(*@KEY@:END_DESCRIPTION*)
FUNCTION_BLOCK V3_SMUL

(*Group:Default*)

VAR_INPUT
	A :	oscat_vector_3;
	M :	REAL;
END_VAR

VAR_OUTPUT
	V3_SMUL :	oscat_vector_3;
END_VAR

(*@KEY@: WORKSHEET
NAME: V3_SMUL
IEC_LANGUAGE: ST
*)
V3_SMUL.X := A.X * M;
V3_SMUL.Y := A.Y * M;
V3_SMUL.Z := A.Z * M;

(* revision history
hm		11 dec 2007	rev 1.0
	original version

*)
(*@KEY@: END_WORKSHEET *)
END_FUNCTION_BLOCK

(* ---- V3_SUB.ST ---- *)
(*@PROPERTIES_EX@
TYPE: POU
LOCALE: 0
IEC_LANGUAGE: ST
PLC_TYPE: independent
PROC_TYPE: independent
GROUP: MATHEMATICAL.VEKTORMATHEMATIK
*)
(*@KEY@:DESCRIPTION*)
version 1.0	11 dec 2007
programmer 	hugo
tested by	tobias

this function subtracts two vectors in a 3 dimensional space
V3_SUB = A - B
(*@KEY@:END_DESCRIPTION*)
FUNCTION_BLOCK V3_SUB

(*Group:Default*)

VAR_INPUT
	A :	oscat_vector_3;
	B :	oscat_vector_3;
END_VAR

VAR_OUTPUT
	V3_SUB :	oscat_vector_3;
END_VAR

(*@KEY@: WORKSHEET
NAME: V3_SUB
IEC_LANGUAGE: ST
*)
V3_SUB.X := A.X - B.X;
V3_SUB.Y := A.Y - B.Y;
V3_SUB.Z := A.Z - B.Z;

(* revision history
hm		11 dec 2007	rev 1.0
	original version

*)
(*@KEY@: END_WORKSHEET *)
END_FUNCTION_BLOCK

(* ---- V3_XANG.ST ---- *)
(*@PROPERTIES_EX@
TYPE: POU
LOCALE: 0
IEC_LANGUAGE: ST
PLC_TYPE: independent
PROC_TYPE: independent
GROUP: MATHEMATICAL.VEKTORMATHEMATIK
*)
(*@KEY@:DESCRIPTION*)
version 1.1	10. mar. 2009
programmer 	hugo
tested by	tobias

this function calculates the angle between the X-axis and a vectors in a 3 dimensional space

(*@KEY@:END_DESCRIPTION*)
FUNCTION_BLOCK V3_XANG

(*Group:Default*)

VAR_INPUT
	A :	oscat_vector_3;
END_VAR

VAR_OUTPUT
	V3_XANG :	REAL;
END_VAR

VAR
	la :	REAL;
	V3_ABS :	V3_ABS;
END_VAR

(*@KEY@: WORKSHEET
NAME: V3_XANG
IEC_LANGUAGE: ST
*)

V3_ABS(A:=A);
la:=V3_ABS.V3_ABS;

IF la > 0.0 THEN
	V3_XANG := ACOS(A.X / la);
ELSE
    V3_XANG := 0.0;
END_IF;

(* revision history
hm	11 dec 2007	rev 1.0
	original version

hm	10. mar. 2009	rev 1.1
	changed syntax of real constants to 0.0

*)
(*@KEY@: END_WORKSHEET *)
END_FUNCTION_BLOCK

(* ---- V3_XPRO.ST ---- *)
(*@PROPERTIES_EX@
TYPE: POU
LOCALE: 0
IEC_LANGUAGE: ST
PLC_TYPE: independent
PROC_TYPE: independent
GROUP: MATHEMATICAL.VEKTORMATHEMATIK
*)
(*@KEY@:DESCRIPTION*)
version 1.0	11 dec 2007
programmer 	hugo
tested by	tobias

this function adds two vectors in a 3 dimensional space
(*@KEY@:END_DESCRIPTION*)
FUNCTION_BLOCK V3_XPRO

(*Group:Default*)

VAR_INPUT
	A :	oscat_vector_3;
	B :	oscat_vector_3;
END_VAR

VAR_OUTPUT
	V3_XPRO :	oscat_vector_3;
END_VAR

(*@KEY@: WORKSHEET
NAME: V3_XPRO
IEC_LANGUAGE: ST
*)
V3_XPRO.X := A.Y * B.Z - A.Z * B.Y;
V3_XPRO.Y := A.Z * B.X - A.X * B.Z;
V3_XPRO.Z := A.X * B.Y - A.Y * B.X;

(* revision history
hm		11 dec 2007	rev 1.0
	original version

*)
(*@KEY@: END_WORKSHEET *)
END_FUNCTION_BLOCK

(* ---- V3_YANG.ST ---- *)
(*@PROPERTIES_EX@
TYPE: POU
LOCALE: 0
IEC_LANGUAGE: ST
PLC_TYPE: independent
PROC_TYPE: independent
GROUP: MATHEMATICAL.VEKTORMATHEMATIK
*)
(*@KEY@:DESCRIPTION*)
version 1.1	10. mar. 2009
programmer 	hugo
tested by	tobias

this function calculates the angle between the Y-axis and a vectors in a 3 dimensional space

(*@KEY@:END_DESCRIPTION*)
FUNCTION_BLOCK V3_YANG

(*Group:Default*)

VAR_INPUT
	A :	oscat_vector_3;
END_VAR

VAR_OUTPUT
	V3_YANG :	REAL;
END_VAR

VAR
	la :	REAL;
	V3_ABS :	V3_ABS;
END_VAR

(*@KEY@: WORKSHEET
NAME: V3_YANG
IEC_LANGUAGE: ST
*)

V3_ABS(A:=A);
la:=V3_ABS.V3_ABS;

IF la > 0.0 THEN
	V3_YANG := ACOS(A.Y / la);
ELSE
    V3_YANG := 0.0;
END_IF;

(* revision history
hm	11 dec 2007	rev 1.0
	original version

hm	10. mar. 2009	rev 1.1
	changed syntax of real constants to 0.0

*)
(*@KEY@: END_WORKSHEET *)
END_FUNCTION_BLOCK

(* ---- V3_ZANG.ST ---- *)
(*@PROPERTIES_EX@
TYPE: POU
LOCALE: 0
IEC_LANGUAGE: ST
PLC_TYPE: independent
PROC_TYPE: independent
GROUP: MATHEMATICAL.VEKTORMATHEMATIK
*)
(*@KEY@:DESCRIPTION*)
version 1.1	10. mar. 2009
programmer 	hugo
tested by	tobias

this function calculates the angle between the Z-axis and a vectors in a 3 dimensional space

(*@KEY@:END_DESCRIPTION*)
FUNCTION_BLOCK V3_ZANG

(*Group:Default*)

VAR_INPUT
	A :	oscat_vector_3;
END_VAR

VAR_OUTPUT
	V3_ZANG :	REAL;
END_VAR

VAR
	la :	REAL;
	V3_ABS :	V3_ABS;
END_VAR

(*@KEY@: WORKSHEET
NAME: V3_ZANG
IEC_LANGUAGE: ST
*)

V3_ABS(A:=A);
la:=V3_ABS.V3_ABS;

IF la > 0.0 THEN
	V3_ZANG := ACOS(A.Z / la);
ELSE
    V3_ZANG := 0.0;
END_IF;

(* revision history
hm	11 dec 2007	rev 1.0
	original version

hm	10. mar. 2009	rev 1.1
	changed syntax of real constants to 0.0

*)
(*@KEY@: END_WORKSHEET *)
END_FUNCTION_BLOCK

(* ---- WEEKDAY_TO_STRING.ST ---- *)
(*@PROPERTIES_EX@
TYPE: POU
LOCALE: 0
IEC_LANGUAGE: ST
PLC_TYPE: independent
PROC_TYPE: independent
GROUP: STRINGS
*)
(*@KEY@:DESCRIPTION*)
version 1.1	19. oct. 2008
programmer 	hugo
tested by	oscat

WEEKDAY_TO_STRING converts an Integer 1..7 into a String with the Names of the corresponding weekday.
the decoding is according to the language setup in global vars
(*@KEY@:END_DESCRIPTION*)
FUNCTION_BLOCK WEEKDAY_TO_STRING

(*Group:Default*)

VAR_INPUT
	WDAY :	INT;
	LANG :	INT;
	LX :	INT;
END_VAR

VAR_OUTPUT
	WEEKDAY_TO_STRING :	oscat_STRING10;
END_VAR

VAR
	LY :	INT;
	SETUP_LANGUAGE :	SETUP_LANGUAGE;
	LANGUAGE :	oscat_LANGUAGE;
	WEEKDAYS :	oscat_WEEKDAYS;
	WEEKDAYS2 :	oscat_WEEKDAYS2;
	SETUP_WEEKDAYS :	SETUP_WEEKDAYS;
	SETUP_WEEKDAYS2 :	SETUP_WEEKDAYS2;
END_VAR

(*@KEY@: WORKSHEET
NAME: WEEKDAY_TO_STRING
IEC_LANGUAGE: ST
*)
SETUP_WEEKDAYS(WEEKDAYS:=WEEKDAYS);
WEEKDAYS:=SETUP_WEEKDAYS.WEEKDAYS;
SETUP_WEEKDAYS2(WEEKDAYS2:=WEEKDAYS2);
WEEKDAYS2:=SETUP_WEEKDAYS2.WEEKDAYS2;
SETUP_LANGUAGE(LANGUAGE:=LANGUAGE);
LANGUAGE:=SETUP_LANGUAGE.LANGUAGE;

IF LANG = 0 THEN ly := LANGUAGE.DEFAULT; ELSE ly := MIN(LANG, LANGUAGE.LMAX); END_IF;
IF wday < 1 OR wday > 7 THEN
	RETURN;
ELSIF LX = 0 THEN
	WEEKDAY_TO_STRING := WEEKDAYS[ly][WDAY];
ELSIF Lx = 2 THEN
	WEEKDAY_TO_STRING := WEEKDAYS2[ly][WDAY];
END_IF;

(* revisison history

hm	21. sep. 2008	rev 1.0
	original version

hm	19. oct. 2008	rev 1.1
	changed language setup constants
*)
(*@KEY@: END_WORKSHEET *)
END_FUNCTION_BLOCK

(* ---- ACOSH.ST ---- *)
(*@PROPERTIES_EX@
TYPE: POU
LOCALE: 0
IEC_LANGUAGE: ST
PLC_TYPE: independent
PROC_TYPE: independent
GROUP: MATHEMATICAL.MATHE
*)
(*@KEY@:DESCRIPTION*)
version 1.3	10. mar. 2009
programmer 	hugo
tested by	tobias

this function calculates the arcus cos hyperbolicus

(*@KEY@:END_DESCRIPTION*)
FUNCTION ACOSH:REAL

(*Group:Default*)

VAR_INPUT
	X :	REAL;
END_VAR

(*@KEY@: WORKSHEET
NAME: ACOSH
IEC_LANGUAGE: ST
*)
ACOSH := LN(SQRT(X * X - 1.0) + X);

(* revision history
hm		12 jan 2007	rev 1.0
	original version

hm		2. dec 2007	rev 1.1
	changed code for better performance

hm	16. mar. 2007		rev 1.2
	changed sequence of calculations to improve performance

hm	10. mar. 2009		rev 1.3
	real constants updated to new systax using dot

*)
(*@KEY@: END_WORKSHEET *)
END_FUNCTION

(* ---- ACOTH.ST ---- *)
(*@PROPERTIES_EX@
TYPE: POU
LOCALE: 0
IEC_LANGUAGE: ST
PLC_TYPE: independent
PROC_TYPE: independent
GROUP: MATHEMATICAL.MATHE
*)
(*@KEY@:DESCRIPTION*)
version 1.2	10. mar. 2009
programmer 	hugo
tested by	tobias

this function calculates the arcus cotangens hyperbolicus

(*@KEY@:END_DESCRIPTION*)
FUNCTION ACOTH:REAL

(*Group:Default*)

VAR_INPUT
	X :	REAL;
END_VAR

(*@KEY@: WORKSHEET
NAME: ACOTH
IEC_LANGUAGE: ST
*)
ACOTH := LN((x+1.0)/(x-1.0))*0.5;

(* revision history
hm		12 jan 2007	rev 1.0
	original version

hm		5. jan 2008	rev 1.1
	improved code for better performance

hm	10. mar. 2009		rev 1.2
	real constants updated to new systax using dot

*)
(*@KEY@: END_WORKSHEET *)
END_FUNCTION

(* ---- AGDF.ST ---- *)
(*@PROPERTIES_EX@
TYPE: POU
LOCALE: 0
IEC_LANGUAGE: ST
PLC_TYPE: independent
PROC_TYPE: independent
GROUP: MATHEMATICAL.MATHE
*)
(*@KEY@:DESCRIPTION*)
version 1.1	10. mar. 2009
programmer 	hugo
tested by	tobias

this function calculates the inverse Gudermannian function.
(*@KEY@:END_DESCRIPTION*)
FUNCTION AGDF:REAL

(*Group:Default*)

VAR_INPUT
	X :	REAL;
END_VAR

(*@KEY@: WORKSHEET
NAME: AGDF
IEC_LANGUAGE: ST
*)
AGDF := LN((1.0 + SIN(X)) / COS(X));

(* comment
the current implementation gives sufficient accuracy only up to X = 1.57 or an output > 10.
is X closer to PI/2 then the function is more and more unreliable
*)

(* revision history
hm	27. apr. 2008	rev 1.0
	original version

hm	10. mar. 2009	rev 1.1
	real constants updated to new systax using dot

*)

(*@KEY@: END_WORKSHEET *)
END_FUNCTION

(* ---- AIN.ST ---- *)
(*@PROPERTIES_EX@
TYPE: POU
LOCALE: 0
IEC_LANGUAGE: ST
PLC_TYPE: independent
PROC_TYPE: independent
GROUP: ENGINEERING.SIGNAL_PROCESSING
*)
(*@KEY@:DESCRIPTION*)
version 1.5	16 mar 2008
programmer 	oscat
tested by	tobias

Ain converts signals from A/D converters or other digital sources to an internal real value
the lowest number of bits are extracted from the input word and the sign will be extracted if available separately.
the output signal is then conditioned to range from low to high values for a 0 to max value on the analog inputs:
for example a 15bit input (bits := 12) with sign at bit 15 (0..15) will deliver 0.0 (low value at 0) for an input value of 2#0000_0000_0000
an input value of 2#1111_1111_1111 will deliver 10.0 on the output (high value set to 10).
(*@KEY@:END_DESCRIPTION*)
FUNCTION AIN:REAL

(*Group:Default*)

VAR_INPUT
	IN :	DWORD;
	BITS :	BYTE;
	SIGN :	BYTE;
	LOW :	REAL;
	HIGH :	REAL;
END_VAR

VAR
	temp1 :	DWORD;
	temp2 :	DWORD;
	sx :	BOOL;
END_VAR

(*@KEY@: WORKSHEET
NAME: AIN
IEC_LANGUAGE: ST
*)
(* extract the sign bit *)
IF sign < BYTE#32 THEN
	temp1 := SHR_DWORD(in, _BYTE_TO_INT(sign));
	sx := BIT_OF_DWORD(temp1,0); (* temp1.X0 *)
ELSE
	sx := FALSE;
END_IF;
temp1 := SHR_DWORD(DWORD#16#FFFFFFFF,32 - _BYTE_TO_INT(bits));
temp2 := in AND temp1;
AIN := (high - low)* _DWORD_TO_REAL(temp2) / _DWORD_TO_REAL(temp1) + low;
IF sx THEN AIN := -AIN; END_IF;

(* revision history
hm 18.8.2006	rev 1.1
	fixed an error with low value negative and high value 0.

hm 19.1.2007	rev 1.2
	fixed an error with sign bit.

hm	13.9.2007	rev 1.3
	changed code to avoid warning under codesys 2.8.1

hm	2. dec 2007	rev 1.4
	changed code for better performance

hm	16. mar 2008	rev 1.5
	added type conversions to avoid warnings under codesys 30
*)
(*@KEY@: END_WORKSHEET *)
END_FUNCTION

(* ---- AOUT.ST ---- *)
(*@PROPERTIES_EX@
TYPE: POU
LOCALE: 0
IEC_LANGUAGE: ST
PLC_TYPE: independent
PROC_TYPE: independent
GROUP: ENGINEERING.SIGNAL_PROCESSING
*)
(*@KEY@:DESCRIPTION*)
version 1.4	23 feb 2008
programmer 	oscat
tested by	tobias

this module conditions an internal real value for D/A converter.
Aout converts and internal real value to a word for an D/A converter or other output devices.
The input value is converted to a n-bit wide output and a sign bit is set separately as specified.
the outout min value is set for the specified min input value and the max output is set for the max input value.
an input higher or lower then the max or min value will set the respective max or min value or the output.
in value or the output.
(*@KEY@:END_DESCRIPTION*)
FUNCTION AOUT:DWORD

(*Group:Default*)

VAR_INPUT
	IN :	REAL;
	BITS :	BYTE;
	SIGN :	BYTE;
	LOW :	REAL;
	HIGH :	REAL;
END_VAR

VAR
	in2 :	REAL;
	sx :	BOOL;
END_VAR

(*@KEY@: WORKSHEET
NAME: AOUT
IEC_LANGUAGE: ST
*)
(* if sign bit is defined *)
IF sign < BYTE#32 THEN
	sx := sign_R(in);
	in2 := ABS(in);
ELSE
	in2 := in;
END_IF;

(* begrenze in auf die zulässigen werte *)
in2 := LIMIT(low, in2, high);

(* Berechne den Ausgangswert *)
Aout := _REAL_TO_DWORD((in2 - low) / (high - low) * (_DWORD_TO_REAL(SHL(DWORD#2#1,_BYTE_TO_INT(bits))) - 1.0)   );
IF sx THEN Aout := SHL_DWORD(DWORD#2#1,_BYTE_TO_INT(sign)) OR Aout; END_IF;

(*
revision history

hm 18.1.2007		rev 1.1
	renamed Modul to aout.
	changed Output to 32 Bit max.
	corrected error with sign bit.

hm	13.9.2007		rev 1.2
	changed code to avoid warning under codesys 2.8.1

hm	2. dec 2007		rev 1.3
	changed code for better performance

hm	23. feb 2008	rev 1.4
	changed code for better performance
*)
(*@KEY@: END_WORKSHEET *)
END_FUNCTION

(* ---- AOUT1.ST ---- *)
(*@PROPERTIES_EX@
TYPE: POU
LOCALE: 0
IEC_LANGUAGE: ST
PLC_TYPE: independent
PROC_TYPE: independent
GROUP: ENGINEERING.SIGNAL_PROCESSING
*)
(*@KEY@:DESCRIPTION*)
version 1.0	23 feb 2008
programmer 	oscat
tested by	tobias

this module conditions an internal real value for a D/A converter.
(*@KEY@:END_DESCRIPTION*)
FUNCTION AOUT1:DWORD

(*Group:Default*)

VAR_INPUT
	IN :	REAL;
	BIT_0 :	INT;
	BIT_N :	INT;
	SIGN :	INT;
	LOW :	REAL;
	HIGH :	REAL;
END_VAR

VAR
	in2 :	REAL;
	sx :	BOOL;
END_VAR

(*@KEY@: WORKSHEET
NAME: AOUT1
IEC_LANGUAGE: ST
*)
(* if sign bit is defined *)

IF sign < 32 THEN
	sx := sign_R(in);
	in2 := ABS(in);
ELSE
    sx := FALSE;
	in2 := in;
END_IF;

(* begrenze in auf die zulässigen werte *)
in2 := LIMIT_REAL(low, in2, high);

(* Berechne den Ausgangswert *)
AOUT1 :=  SHL_DWORD(_REAL_TO_DWORD((in2 - low) / (high - low) * UDINT_TO_REAL(DWORD_TO_UDINT(SHL(DWORD#2#1,bit_n - Bit_0 + 1)) - UDINT#1)),Bit_0);

IF sx THEN AOUT1 := SHL(DWORD#2#1,sign) OR AOUT1; END_IF;

(* revision history
hm	23. feb 2008	rev 1.0
	original version

*)
(*@KEY@: END_WORKSHEET *)
END_FUNCTION

(* ---- ASINH.ST ---- *)
(*@PROPERTIES_EX@
TYPE: POU
LOCALE: 0
IEC_LANGUAGE: ST
PLC_TYPE: independent
PROC_TYPE: independent
GROUP: MATHEMATICAL.MATHE
*)
(*@KEY@:DESCRIPTION*)
version 1.3	10. mar 2009
programmer 	hugo
tested by	tobias

this function calculates the arcus sin hyperbolicus
(*@KEY@:END_DESCRIPTION*)
FUNCTION ASINH:REAL

(*Group:Default*)

VAR_INPUT
	X :	REAL;
END_VAR

(*@KEY@: WORKSHEET
NAME: ASINH
IEC_LANGUAGE: ST
*)
ASINH := LN(SQRT(X * X + 1.0)+X);

(* revision history
hm		12 jan 2007	rev 1.0
	original version

hm		2. dec 2007	rev 1.1
	changed code for better performance

hm		16.3. 2007		rev 1.2
	changed sequence of calculations to improve performance

hm	10. mar. 2009		rev 1.3
	real constants updated to new systax using dot

*)
(*@KEY@: END_WORKSHEET *)
END_FUNCTION

(* ---- ATAN2.ST ---- *)
(*@PROPERTIES_EX@
TYPE: POU
LOCALE: 0
IEC_LANGUAGE: ST
PLC_TYPE: independent
PROC_TYPE: independent
GROUP: MATHEMATICAL.MATHE
*)
(*@KEY@:DESCRIPTION*)
version 1.2	10. mar. 2009
programmer 	hugo
tested by	oscat

this function calculates the angle in a coordinate system in rad.
(*@KEY@:END_DESCRIPTION*)
FUNCTION ATAN2:REAL

(*Group:Default*)

VAR_INPUT
	X :	REAL;
	Y :	REAL;
END_VAR

(*@KEY@: WORKSHEET
NAME: ATAN2
IEC_LANGUAGE: ST
*)
IF X > 0.0 THEN
	ATAN2 := ATAN(Y/X);
ELSIF X < 0.0 THEN
	IF Y >= 0.0 THEN
		ATAN2 := ATAN(Y/X) + 3.14159265358979323846264338327950288;
	ELSE
		ATAN2 := ATAN(Y/X) - 3.14159265358979323846264338327950288;
	END_IF;
ELSIF Y > 0.0 THEN
	ATAN2 := 1.5707963267948965580;
ELSIF Y < 0.0 THEN
	ATAN2 := -1.5707963267948965580;
ELSE
	ATAN2 := 0.0;
END_IF;

(* revision history
hm	20.  apr. 2008	rev 1.0
	original version

hm	18. oct. 2008	rev 1.1
	changed to use math constants

hm	10. mar. 2009	rev 1.2
	real constants updated to new systax using dot

*)
(*@KEY@: END_WORKSHEET *)
END_FUNCTION

(* ---- ATANH.ST ---- *)
(*@PROPERTIES_EX@
TYPE: POU
LOCALE: 0
IEC_LANGUAGE: ST
PLC_TYPE: independent
PROC_TYPE: independent
GROUP: MATHEMATICAL.MATHE
*)
(*@KEY@:DESCRIPTION*)
version 1.2	10. mar. 2009
programmer 	hugo
tested by	tobias

this function calculates the arcus tangens hyperbolicus
(*@KEY@:END_DESCRIPTION*)
FUNCTION ATANH:REAL

(*Group:Default*)

VAR_INPUT
	X :	REAL;
END_VAR

(*@KEY@: WORKSHEET
NAME: ATANH
IEC_LANGUAGE: ST
*)
ATANH := LN((1.0 + x)/(1.0 - x)) * 0.5;

(* revision history
hm		12 jan 2007	rev 1.0
	original version

hm		5. jan 2008	rev 1.1
	improved code for better performance

hm	10. mar. 2009		rev 1.2
	real constants updated to new systax using dot

*)
(*@KEY@: END_WORKSHEET *)
END_FUNCTION

(* ---- BAND_B.ST ---- *)
(*@PROPERTIES_EX@
TYPE: POU
LOCALE: 0
IEC_LANGUAGE: ST
PLC_TYPE: independent
PROC_TYPE: independent
GROUP: ENGINEERING.CONTROL
*)
(*@KEY@:DESCRIPTION*)
version 1.0	21. Nov. 2008
programmer 	hugo
tested by	oscat

BAND_B will limit X to B <= X <= 255-B. while X < B the resulkt will be 0 and while X > 255-B the output will be 255
otherwise the result = X.
(*@KEY@:END_DESCRIPTION*)
FUNCTION BAND_B:BYTE

(*Group:Default*)

VAR_INPUT
	X :	BYTE;
	B :	BYTE;
END_VAR

(*@KEY@: WORKSHEET
NAME: BAND_B
IEC_LANGUAGE: ST
*)
IF X < B THEN
	BAND_B := BYTE#0;
ELSIF X > USINT_TO_BYTE(USINT#255 - BYTE_TO_USINT(B)) THEN
	BAND_B := BYTE#255;
ELSE
	BAND_B := X;
END_IF;

(* revision history
hm	21. nov. 2008	rev 1.0
	original version

*)
(*@KEY@: END_WORKSHEET *)
END_FUNCTION

(* ---- BCDC_TO_INT.ST ---- *)
(*@PROPERTIES_EX@
TYPE: POU
LOCALE: 0
IEC_LANGUAGE: ST
PLC_TYPE: independent
PROC_TYPE: independent
GROUP: LOGIC.GATE_LOGIC
*)
(*@KEY@:DESCRIPTION*)
version 1.1	30. jun. 2008
programmer 	hugo
tested by	tobias

this function converts a two digit bcd number into an integer.
(*@KEY@:END_DESCRIPTION*)
FUNCTION BCDC_TO_INT:INT

(*Group:Default*)

VAR_INPUT
	IN :	BYTE;
END_VAR

(*@KEY@: WORKSHEET
NAME: BCDC_TO_INT
IEC_LANGUAGE: ST
*)
BCDC_TO_INT := _BYTE_TO_INT(in AND BYTE#16#0F) + (_BYTE_TO_INT(SHR(in,4)) * 10);

(* revision history
hm	13.12.2007		rev 1.0
	original version

hm	30. jun. 2008	rev 1.1
	changed name to avoid collision with util.lib
*)
(*@KEY@: END_WORKSHEET *)
END_FUNCTION

(* ---- BETA.ST ---- *)
(*@PROPERTIES_EX@
TYPE: POU
LOCALE: 0
IEC_LANGUAGE: ST
PLC_TYPE: independent
PROC_TYPE: independent
GROUP: MATHEMATICAL.MATHE
*)
(*@KEY@:DESCRIPTION*)
version 1.0	26. oct. 2008
programmer 	hugo
tested by	oscat

this function calculates the beta function for real number > 0.
(*@KEY@:END_DESCRIPTION*)
FUNCTION BETA:REAL

(*Group:Default*)

VAR_INPUT
	X :	REAL;
	Y :	REAL;
END_VAR

(*@KEY@: WORKSHEET
NAME: BETA
IEC_LANGUAGE: ST
*)
BETA := GAMMA(X)*GAMMA(Y) / GAMMA(x+y);

(* revision history
hm	26. oct. 2008	rev 1.0
	original version

*)
(*@KEY@: END_WORKSHEET *)
END_FUNCTION

(* ---- BFT_TO_MS.ST ---- *)
(*@PROPERTIES_EX@
TYPE: POU
LOCALE: 0
IEC_LANGUAGE: ST
PLC_TYPE: independent
PROC_TYPE: independent
GROUP: ENGINEERING.CONVERSION
*)
(*@KEY@:DESCRIPTION*)
version 1.0	12. jun 2008
programmer 	hugo
tested by	oscdat

this function converts wind speed from beaufort to m/s
(*@KEY@:END_DESCRIPTION*)
FUNCTION BFT_TO_MS:REAL

(*Group:Default*)

VAR_INPUT
	BFT :	INT;
END_VAR

(*@KEY@: WORKSHEET
NAME: BFT_TO_MS
IEC_LANGUAGE: ST
*)
BFT_TO_MS := EXPT(INT_TO_REAL(BFT), 1.5) * 0.836;

(* revision history
hm	12. 6. 2008		rev 1.0
	original version

*)
(*@KEY@: END_WORKSHEET *)
END_FUNCTION

(* ---- BINOM.ST ---- *)
(*@PROPERTIES_EX@
TYPE: POU
LOCALE: 0
IEC_LANGUAGE: ST
PLC_TYPE: independent
PROC_TYPE: independent
GROUP: MATHEMATICAL.MATHE
*)
(*@KEY@:DESCRIPTION*)
version 1.0	25. oct. 2008
programmer 	hugo
tested by	tobias

this function calculates the binomialkoefficient (N over k)
(*@KEY@:END_DESCRIPTION*)
FUNCTION BINOM:INT

(*Group:Default*)

VAR_INPUT
	N :	INT;
	K :	INT;
END_VAR

VAR
	i :	INT;
	N2 :	INT;
	K2 :	INT;
END_VAR

(*@KEY@: WORKSHEET
NAME: BINOM
IEC_LANGUAGE: ST
*)
K2 := K;
N2 := N;
IF 2 * K2 > N2 THEN
	K2 := N2 - K2;
END_IF;
IF K2 > N2 THEN
	RETURN;
ELSIF K2 = 0 OR K2 = N2 THEN
	BINOM := 1;
ELSIF K2 = 1 THEN
	BINOM := N2;
ELSE
	BINOM := N2;
	N2 := N2 + 1;
	FOR i := 2 TO K2 DO
		BINOM := BINOM * (N2 - i) / i;
	END_FOR;
END_IF;

(*
binomialkoeffizient(n, k)
1  wenn k = 0 return 1
2  wenn 2k > n
3      dann führe aus ergebnis \leftarrow binomialkoeffizient(n, n-k)
4  sonst führe aus ergebnis \leftarrow n
5          von i \leftarrow 2 bis k
6              führe aus ergebnis \leftarrow ergebnis \cdot (n + 1 - i)
7                        ergebnis \leftarrow ergebnis : i
8  return ergebnis
*)

(* revision history
hm	25. oct. 2008	rev 1.0
	original version

*)
(*@KEY@: END_WORKSHEET *)
END_FUNCTION

(* ---- BIT_COUNT.ST ---- *)
(*@PROPERTIES_EX@
TYPE: POU
LOCALE: 0
IEC_LANGUAGE: ST
PLC_TYPE: independent
PROC_TYPE: independent
GROUP: LOGIC.GATE_LOGIC
*)
(*@KEY@:DESCRIPTION*)
version 1.1	10 sep 2007
programmer 	hugo
tested by	tobias

BIT_COUNT counts the amount True of bits in a dword.
for exabple: bit_count(3) returns 2 because two bits (bits 0 and 1) are true and all others are false.
(*@KEY@:END_DESCRIPTION*)
FUNCTION BIT_COUNT:INT

(*Group:Default*)

VAR_INPUT
	IN :	DWORD;
END_VAR

VAR
	in_temp :	DWORD;
END_VAR

(*@KEY@: WORKSHEET
NAME: BIT_COUNT
IEC_LANGUAGE: ST
*)
in_temp := IN;
WHILE in_temp > DWORD#0 DO
	IF (in_temp AND DWORD#16#00000001) > DWORD#0 THEN Bit_Count := Bit_Count +1; END_IF;
	in_temp := SHR(in_temp,1);
END_WHILE;

(* revision history
5.7.2007	rev 1.0		original version

10.9.2007	rev 1.1		hm
	changed algorithm for better performace
	the execution time has reduced by a factor of 5
	deleted unused variable temp
*)
(*@KEY@: END_WORKSHEET *)
END_FUNCTION

(* ---- BIT_LOAD_B.ST ---- *)
(*@PROPERTIES_EX@
TYPE: POU
LOCALE: 0
IEC_LANGUAGE: ST
PLC_TYPE: independent
PROC_TYPE: independent
GROUP: LOGIC.GATE_LOGIC
*)
(*@KEY@:DESCRIPTION*)
version 1.1	16. mar 2008
programmer 	hugo
tested by	tobias

this function loads a bit into a byte at position pos.
(*@KEY@:END_DESCRIPTION*)
FUNCTION BIT_LOAD_B:BYTE

(*Group:Default*)

VAR_INPUT
	IN :	BYTE;
	VAL :	BOOL;
	POS :	INT;
END_VAR

(*@KEY@: WORKSHEET
NAME: BIT_LOAD_B
IEC_LANGUAGE: ST
*)
IF VAL THEN
	BIT_LOAD_B := in OR SHL(BYTE#1,pos);
ELSE
	BIT_LOAD_B := in AND (NOT SHL(BYTE#1,pos));
END_IF;

(* revision history
hm	29. feb 2008	rev 1.0
	original version

hm	16. mar 2008	rev 1.1
	change input bit to val for compatibility reasons
*)
(*@KEY@: END_WORKSHEET *)
END_FUNCTION

(* ---- BIT_LOAD_B2.ST ---- *)
(*@PROPERTIES_EX@
TYPE: POU
LOCALE: 0
IEC_LANGUAGE: ST
PLC_TYPE: independent
PROC_TYPE: independent
GROUP: LOGIC.GATE_LOGIC
*)
(*@KEY@:DESCRIPTION*)
version 1.0 18. oct. 2008
programmer 	hugo
tested by	tobias

this function loads N bits of D at pos P in Byte I
(*@KEY@:END_DESCRIPTION*)
FUNCTION BIT_LOAD_B2:BYTE

(*Group:Default*)

VAR_INPUT
	I :	BYTE;
	D :	BOOL;
	P :	INT;
	N :	INT;
END_VAR

(*@KEY@: WORKSHEET
NAME: BIT_LOAD_B2
IEC_LANGUAGE: ST
*)
IF D THEN
	BIT_LOAD_B2 := ROL(SHR(BYTE#255, 8 - N) OR ROR(I, P), P);
ELSE
	BIT_LOAD_B2 := ROL(SHL(BYTE#255, N) AND ROR(I, P), P);
END_IF;

(* revision history
hm	18. oct. 2008	rev 1.0
	original version

*)
(*@KEY@: END_WORKSHEET *)
END_FUNCTION
